(* CODESYS project twincat3_dioc_lib.library
   Author: AH
   Placeholder: Dioc
   Title: DiocLibrary
   Version: 3.25
   Company: Upzio

Project tree, tasks and I/O mapping:
  libraries: Tc2_Standard, * (Beckhoff Automation GmbH); Tc2_System, * (Beckhoff Automation GmbH); Tc2_Utilities, * (Beckhoff Automation GmbH); VisuDialogs, * (System)
  Data types/
    DIOC/
      Dioc/
        data type A_DIOC_DATA_TYPE
        data type A_DIOC_DATA_TYPE_1
        data type A_DIOC_MESSAGE
        data type A_DIOC_REGISTER_TYPE
        data type E_DIOC_ERROR
        data type E_DIOC_GEN_ERROR
        data type E_DIOC_REGISTER
        data type E_SM_DIOC
        data type E_SM_DIOC_DEVICE
        data type E_SM_DIOC_RECEIVE
        data type E_SM_DIOC_SEND
        data type ST_DIOC
        data type ST_DIOC_GEN_IN
        data type ST_DIOC_GEN_OUT
        data type ST_DIOC_IN
        data type ST_DIOC_LOG
        data type ST_DIOC_MESSINFO
        data type ST_DIOC_OUT
        data type ST_DIOC_REGISTER
      RC/
        RC/
          data type E_DIOC_RC_ERROR
          data type E_DIOC_RC_REGISTER
          data type E_RC_ERROR
          data type ST_DIOC_RC_IN
          data type ST_DIOC_RC_OUT
          data type ST_RC_IN
          data type ST_RC_OUT
      TP/
        TP10/
          data type E_DIOC_TP10_ERROR
          data type E_DIOC_TP10_REGISTER
          data type E_TP10
          data type E_TP10_ERROR
          data type ST_DIOC_TP10_IN
          data type ST_DIOC_TP10_OUT
          data type ST_TP10_IN
          data type ST_TP10_OUT
  Global Variables/
    global variables Global_DIOC_Constants
    global variables Global_DIOC_Variables
    global variables Global_DIOC_Variables_Debug
  POUs/
    DIOC/
      _Internal/
        DIOC/
          Dioc20/
            function F_DIOC_20_MESSAGE_IN [ST]
            function F_DIOC_20_MESSAGE_OUT [ST]
          function block FB_DIOC [ST]: Receive, Send, Startup
          function block FB_DIOC_GEN [ST]: Receive, Reset, Restart, Send, Startup
        DIOC_HELPFUNCTIONS/
          function F_DIOC_INC2 [ST]
          function F_DIOC_TO_DATE [ST]
          function F_SCALE_FROM_DIOC [ST]
          function F_SCALE_FROM_DIOC_FO [ST]
          function F_SCALE_FROM_REAL [ST]
          function F_SCALE_TO_DIOC [ST]
          function block FB_DIOC_FIFO [ST]
          function block FB_DIOC_RING [ST]
          function block FB_DIOC_RING2 [ST]
      RC/
        _Internal/
          function block FB_DIOC_RC [ST]: Receive, Restart, Send, Startup
          function block FB_RC_COMM [ST]: Startup
        function block FB_RC [ST]: StartupList, Stateinit
      TP10/
        _Internal/
          function block FB_DIOC_TP10 [ST]: Receive, Restart, Send, Startup
          function block FB_TP10_COMM [ST]: Startup
        function block FB_TP10 [ST]: StartupList, Stateinit
      function F_GetVersion_FIXSUS_DIOC [ST]
  Visualizations/
    DIOC/
      RC/
        RC_PARTS/
          visualisation RC_FP
          visualisation RC_ROOM_ICON
          visualisation UDO_DIPSWITCH
        visualisation RC
        visualisation RC_MINI
      TP10/
        TP10_PARTS/
          visualisation TP10_FP
          visualisation TP10_ROOM_ICON
        visualisation TP10
        visualisation TP10_MINI
  GlobalImagePool
*)

// Data types/DIOC/Dioc/A_DIOC_DATA_TYPE
TYPE A_DIOC_DATA_TYPE : DWORD;
END_TYPE

// Data types/DIOC/Dioc/A_DIOC_DATA_TYPE_1
TYPE A_DIOC_DATA_TYPE_1 : DWORD;
END_TYPE

// Data types/DIOC/Dioc/A_DIOC_MESSAGE
TYPE A_DIOC_MESSAGE : DWORD;
END_TYPE

// Data types/DIOC/Dioc/A_DIOC_REGISTER_TYPE
TYPE A_DIOC_REGISTER_TYPE : INT;
END_TYPE

// Data types/DIOC/Dioc/E_DIOC_ERROR
TYPE E_DIOC_ERROR :
(
	DIOC_ERROR_NO_ERROR
);
END_TYPE

// Data types/DIOC/Dioc/E_DIOC_GEN_ERROR
TYPE E_DIOC_GEN_ERROR :
(
	DIOC_REG_ERROR_NO_ERROR,
	DIOC_REG_ERROR_WRONG_TYPEID
);
END_TYPE

// Data types/DIOC/Dioc/E_DIOC_REGISTER
TYPE E_DIOC_REGISTER :
(
	DIOC_R00_SYNC_MESSAGE				:= 0,
	DIOC_R01_REGISTER_REQUEST			:= 1,
	DIOC_R02_REGISTER_INTERVAL			:= 2,
	DIOC_R03_TYPE_ID					:= 3,
	DIOC_R04_VERSION_HW					:= 4,
	DIOC_R05_VERSION_SW					:= 5,
	DIOC_R06_VERSION_REGISTERS			:= 6,
	DIOC_R07_UNIQUE_ID					:= 7,
	DIOC_R08_MESSAGE_ERROR_COUNTER		:= 8,
	DIOC_R09_VOLTAGE_LEVEL_A			:= 9,
	DIOC_R10_VOLTAGE_LEVEL_B			:= 10,
	DIOC_R11_DEVICE_ENABLE				:= 11,
	DIOC_R12_CPU_TEMPERATURE			:= 12,
	DIOC_R13_ErrorRegisterAdress		:= 13,

	DIOC_R84_TRANSMIT_DELAY				:= 84,
	DIOC_R85_SYNC_MESSAGE_HIGH			:= 85
);
END_TYPE

// Data types/DIOC/Dioc/E_SM_DIOC
TYPE E_SM_DIOC :
(
	SM_DIOC_POWERUP_DEVICE,					(* Activate device *)
	SM_DIOC_WAIT_FOR_DEVICE_CHARGED,		(* Activation timer, can be deactivated *)
	SM_DIOC_SEND_SYNC_REQUEST,				(* sync request by master *)
	SM_DIOC_WAIT_FOR_SYNC_ACK,				(* sync acknowledge by device *)
	SM_DIOC_SEND_SYNC_ACK,					(* sync acknowledge by master *)
	SM_DIOC_SEND_STARTUP_VALUES,			(* OPTIONAL Send optional startup values *)
	SM_DIOC_SEND_NEXTSTARTUP_VALUES,		(* OPTIONAL Send optional startup values *)
	SM_DIOC_R11_DEVICE_ENABLE,				(* OPTIONAL Enable Device *)
	SM_DIOC_R11_DEVICE_ENABLED,				(* OPTIONAL Enable Device *)
	SM_DIOC_ACTIVE				:= 100,		(* device is active *)
	SM_DIOC_END,
	SM_DIOC_TEST,
	SM_DIOC_WAIT_FOR_RESTART,				(* Delay time to restart after device failure *)
	SM_DIOC_ERROR 				:=666
);
END_TYPE

// Data types/DIOC/Dioc/E_SM_DIOC_DEVICE
TYPE E_SM_DIOC_DEVICE :
(
	SM_DIOC_DEVICE_POWERUP_DEVICE,					(* Power up device *)
	SM_DIOC_DEVICE_SEND_SYNC_REQUEST,				(* sync message by master *)
	SM_DIOC_DEVICE_SEND_SECOND_SYNC_REQUEST,		(* sync request by master *)
	SM_DIOC_DEVICE_WAIT_FOR_TYPE_ID,				(* wait until the device sent it's type id *)
	SM_DIOC_DEVICE_SEND_SYNC_ACK,					(* sync acknowledge by master *)
	SM_DIOC_DEVICE_SEND_STARTUP_VALUES,				(* OPTIONAL Send optional startup values *)
	SM_DIOC_DEVICE_STARTUP_VALUES_SENT,				(* OPTIONAL startup values sent *)
	SM_DIOC_DEVICE_DEVICE_ENABLE,					(* OPTIONAL Enable Device *)
	SM_DIOC_DEVICE_DEVICE_ENABLED,					(* OPTIONAL Enable Device *)
	SM_DIOC_DEVICE_RESTART,							(* device was restarted, wait until alle settings are re-written *)
	SM_DIOC_DEVICE_ACTIVE					:= 100,	(* device is active *)
	SM_DIOC_DEVICE_END,
	SM_DIOC_DEVICE_TEST,
	SM_DIOC_DEVICE_ERROR 					:= 666
);
END_TYPE

// Data types/DIOC/Dioc/E_SM_DIOC_RECEIVE
TYPE E_SM_DIOC_RECEIVE :
(
	SM_DIOC_RECEIVE_WAIT_FOR_DEVICE,
	SM_DIOC_RECEIVE_WAIT_FOR_STARTBIT,
	SM_DIOC_RECEIVE_RECEIVE_BITS,
	SM_DIOC_RECEIVE_WAIT_FOR_BUFFER,
	SM_DIOC_RECEIVE_END,
	SM_DIOC_RECEIVE_TEST,
	SM_DIOC_RECEIVE_ERROR	:= 666
);
END_TYPE

// Data types/DIOC/Dioc/E_SM_DIOC_SEND
TYPE E_SM_DIOC_SEND :
(
	SM_DIOC_SEND_WAIT_FOR_DEVICE,
	SM_DIOC_SEND_START,
	SM_DIOC_SEND_BITS,
	SM_DIOC_SEND_END,
	SM_DIOC_SEND_TEST,
	SM_DIOC_SEND_ERROR 			:=666
);
END_TYPE

// Data types/DIOC/Dioc/ST_DIOC
TYPE ST_DIOC :
STRUCT
	in						: ST_DIOC_IN;
	out						: ST_DIOC_OUT;
END_STRUCT
END_TYPE

// Data types/DIOC/Dioc/ST_DIOC_GEN_IN
TYPE ST_DIOC_GEN_IN :
STRUCT
	(* COMMANDS to device, bit reset by device block as an acknowledge *)
	(*Send start parameter*)

	bRxx_StartPar						: BOOL;

	(* Send test message *)
	bRxx_SendMessage					: BOOL;
	(* Send sync message *)
	bR00_SyncMessage					: BOOL;
	(* Register 1 / 2: register request *)
	bR01_RegisterRequest				: BOOL;
	bR01_RegisterRequestAutoSend		: BOOL;
	(* Sync delay *)
	bR84_TransmitDelay_READ				: BOOL;
	bR84_TransmitDelay_WRITE			: BOOL;

	(* COMMANDS to device, device uses the bit but does not alter it, eg output is switched when bit high, switched off when bit low *)
	bR03_Request_Type_ID				: BOOL;						(* R03: Type ID of the device *)
	bR04_Request_HW_Version				: BOOL;						(* R04: Hardware version of the device *)
	bR05_Request_SW_Version				: BOOL;						(* R05: Software version of the device *)
	bR06_Request_Register_Version		: BOOL;						(* R06: Register version of the device *)
	bR07_Request_Unique_ID				: BOOL;						(* R07: Unique ID of the device *)
	bR08_Message_Error_Counter_READ		: BOOL;						(* R08: message error counter *)
	bR08_Message_Error_Counter_WRITE	: BOOL;						(* R08: message error counter reset *)
	bR09_Read_DiocA_Voltage_Level		: BOOL;						(* R09: Read DIOCA voltage level (x10) *)
	bR10_Read_DiocB_Voltage_Level		: BOOL;						(* R10: Read DIOCB voltage level (x10) *)
	bR11_Enable_Device_READ				: BOOL;						(* R11: Device Enable *)
	bR11_Enable_Device					: BOOL;						(* R11: Device Enable *)
	bR11_Disable_Device					: BOOL;						(* R11: Device Disable *)
	bR12_CPU_Temperature				: BOOL;						(* R12: CPU Temperature *)

	(* DIOC OUTPUT PARAMETERS, parameters necessary for the above commands *)
	(* Send test message *)
	byRxx_SendMessageRegister 			: A_DIOC_REGISTER_TYPE	;	(* register address not inverted *)
	dwRxx_SendMessageData 				: A_DIOC_DATA_TYPE	:= 2#10;		(* data not inverted *)
	(* Register 1 / 2: register request *)
	dwR01_MessageRegister 				: A_DIOC_DATA_TYPE	;	(* register address not inverted *)
	dwR02_MessageAutoSendInterval		: A_DIOC_DATA_TYPE	:= 0;	(* 10 bit in seconds *)
	nR08_MessageErrorCounter			: UINT := 0;				(* R8: Message Err. Counter, onnly to be set <> 0 for unittest *)
	(* Sync delay *)
	dwR84_TransmitDelay					: A_DIOC_DATA_TYPE;
END_STRUCT
END_TYPE

// Data types/DIOC/Dioc/ST_DIOC_GEN_OUT
TYPE ST_DIOC_GEN_OUT :
STRUCT
	bDeviceActive					: BOOL;						(* Device is active *)
	(* Buffer statusses
	bRxBufferEmpty					: BOOL;						(* RX Buffer empty *)
	bRxBufferFull					: BOOL;						(* RX Buffer full *)
	bTxBufferEmpty					: BOOL;						(* All TX Buffer empty *)
	bTxBufferFull					: BOOL;						(* At least 1 TX Buffer full *)*)

	(* Internal feedback *)
	bTEST_LastMessageOK_Test		: BOOL;
	bRxx_Received					: BOOL;						(* There was a new message from the device *)

	(* RC register feedback bits *)
	bR11_DeviceEnabled				: BOOL;						(* R11: Device Enable *)

	(* RC register feedback values *)
	nRxx_Received					: INT;						(* There was a new message from the device from this register *)
	nR03_TypeID						: INT;						(* R3: Type ID *)
	nR08_MessageErrorCounter		: UINT;						(* R8: Message Err. Counter *)
	nR09_DiocVoltageA				: REAL := -3.402823E38; 	(* R9: Read DIOCA voltage level (x10) *)
	nR10_DiocVoltageB				: REAL := -3.402823E38; 	(* R10: Read DIOCA voltage level (x10) *)
	nR12_CpuTemperature				: REAL := -3.402823E38; 	(* R12: CPU Temperature *)
	nR13_ErrorRegisterAdress		: UINT;
	sR13_DtLastError				: STRING;
	nR84_TransmitDelay				: REAL := -3.402823E38;		(* R84: 'transmit delay (timeshift PLC<-> device) *)
	dtR04_VersionHW					: DATE;						(* R4: Version HW, 7 scrolls *)
	dtR05_VersionSW					: DATE;						(* R5: Version SW, 7 scrolls *)
	dtR06_VersionREG				: DATE;						(* R6: Version Registers, 7 scrolls *)
	sR07_UniqueID					: STRING[24];				(* R7: Unique ID *)
END_STRUCT
END_TYPE

// Data types/DIOC/Dioc/ST_DIOC_IN
TYPE ST_DIOC_IN :
STRUCT
	bEnable					: BOOL := TRUE;			(* TRUE powers the device *)
END_STRUCT
END_TYPE

// Data types/DIOC/Dioc/ST_DIOC_LOG
TYPE ST_DIOC_LOG :
STRUCT
	Message:ST_DIOC_REGISTER;
	Timestamp:DT;
	iArrId:INT;
END_STRUCT
END_TYPE

// Data types/DIOC/Dioc/ST_DIOC_MESSINFO
TYPE ST_DIOC_MESSINFO :
STRUCT
	nRegister							: A_DIOC_REGISTER_TYPE;
	nValue								: A_DIOC_DATA_TYPE;
	dt_Time								: DATE_AND_TIME;
	ArrnumberDIOC						: INT;
	iErrCode							: INT;
	iDeviceType							: INT;
END_STRUCT
END_TYPE

// Data types/DIOC/Dioc/ST_DIOC_OUT
TYPE ST_DIOC_OUT :
STRUCT
	bDeviceReady					: BOOL;				(* Device charged and ready *)
	(* DIOC Buffer statusses *)
	bRxBufferEmpty					: BOOL;				(* RX Buffer empty *)
	bRxBufferFull					: BOOL;				(* RX Buffer full *)
	bTxBufferEmpty					: BOOL;				(* All TX Buffer empty *)
	bTxBufferFull					: BOOL;				(* At least 1 TX Buffer full *)
	bBusyReceiving					: BOOL;			(* Receiving new data  *)
	bBusySending					: BOOL;				(* Sending data *)
	bError							: BOOL;				(* Dioc error state *)
	nErrorID						: E_DIOC_ERROR;		(* Dioc error code *)
	dwDataReceived					: DWORD;			(* Data received *)
END_STRUCT
END_TYPE

// Data types/DIOC/Dioc/ST_DIOC_REGISTER
TYPE ST_DIOC_REGISTER :
STRUCT
	nPLC_Cycle			: WORD;		(* Only for debugging *)
	nRegister			: A_DIOC_REGISTER_TYPE;
	nValue				: A_DIOC_DATA_TYPE;
END_STRUCT
END_TYPE

// Data types/DIOC/RC/RC/E_DIOC_RC_ERROR
TYPE E_DIOC_RC_ERROR :
(
	DIOC_RC_ERROR_NO_ERROR
);
END_TYPE

// Data types/DIOC/RC/RC/E_DIOC_RC_REGISTER
TYPE E_DIOC_RC_REGISTER :
(
	RC_R20_RC_TEMPERATURE			:= 20,
	RC_R21_PS_AC_VOLTAGE_LEVEL,
	RC_R22_STATUS_BITS_DIPSWITCHES,
	RC_R25_HEATING_7_8_3P			:= 25,
	RC_R26_HEATING_9_SP,
	RC_R27_HEATING_12_13_TEMP_HVAC_WATER,
	RC_R32_COOLING_20_21_3P		:= 32,
	RC_R33_COOLING_22_SP,
	RC_R34_COOLING_25_26_TEMP_ICE_WATER,
	RC_R39_PULSION_16_POSITION_COMMAND := 39,
	RC_R40_PULSION_17_POSITION_FEEDBACK,
	RC_R42_PULSION_18_AIR_TEMPERATURE := 42,
	RC_R45_EXTRACTION_29_POSITION_COMMAND := 45,
	RC_R46_EXTRACTION_30_POSITION_FEEDBACK,
	RC_R49_EXTRACTION_31_AIR_TEMPERATURE := 49,
	RC_R52_FIREDAMPER_33_34_COMMAND := 52,
	RC_R53_FIREDAMPER_36_37_FEEDBACK,
	RC_R56_FAN_39_40_SPEED_COMMAND 	:= 56,
	RC_R57_FAN_ENABLE,
	RC_R58_FAN_FAULT_STATUS,
	RC_R61_DO_45_46_47				:= 61,

	RC_R82_temperature_readout_adjust	:= 82,
	RC_R84_TRANSMIT_DELAY				:= 84,
	RC_R85_SYNC_MESSAGE_HIGH			:= 85
);
END_TYPE

// Data types/DIOC/RC/RC/E_RC_ERROR
TYPE E_RC_ERROR :
(
	RC_ERROR_NO_ERROR
);
END_TYPE

// Data types/DIOC/RC/RC/ST_DIOC_RC_IN
TYPE ST_DIOC_RC_IN :
STRUCT
	(* Startup list *)
	arrstStartupParameter				: ARRAY[1..DIOC_NOOFSTARTUPPARAMETERS] OF ST_DIOC_REGISTER;

	bR20_RC_Temperature				: BOOL;						(* R20: RC Temperature *)
	bR21_Read_PS_AC_Voltage				: BOOL;						(* R21: Read PS AC voltage level (x10) *)
	bR22_Status_Dip_Switches			: BOOL;						(* R22: Status bits DIP switches *)
	bR23_reserve						: BOOL;
	bR24_reserve						: BOOL;
	bR25_Heating_7_8_3p_plus_pwm		: BOOL;						(* R25: Heating 7-8 bit 0: 3p+/pwm, bit 1: 3p- *)
	bR25_Heating_7_8_3p_min				: BOOL;						(* R25: Heating 7-8 bit 0: 3p+/pwm, bit 1: 3p- *)
	bR25_Heating_7_8_3p_status			: BOOL;						(* R25: Heating 7-8 bit 0: 3p+/pwm, bit 1: 3p- *)
	bR26_Heating_SP						: BOOL;						(* R26: Heating 9  SP 0..10V *)
	bR26_Heating_SP_status				: BOOL;						(* R26: Heating 9  SP 0..10V *)
	bR27_Heating_T						: BOOL;						(* R27: Heating 12-13 temperature HVAC water *)
	bR28_reserve						: BOOL;
	bR29_reserve						: BOOL;
	bR30_reserve						: BOOL;
	bR31_reserve						: BOOL;
	bR32_Cooling_20_21_3p_plus_pwm		: BOOL;						(* R32: Cooling 20-21 bit 0: 3p+/pwm   1: 3p- *)
	bR32_Cooling_20_21_3p_min			: BOOL;						(* R32: Cooling 20-21 bit 0: 3p+/pwm   1: 3p- *)
	bR32_Cooling_20_21_3p_status		: BOOL;						(* R32: Cooling 20-21 bit 0: 3p+/pwm   1: 3p- *)
	bR33_Cooling_SP						: BOOL;						(* R33: Cooling 22  SP 0..10V *)
	bR33_Cooling_SP_status				: BOOL;						(* R33: Cooling 22  SP 0..10V *)
	bR34_Cooling_T						: BOOL;						(* R34: Cooling 25-26 temperature ICE water *)
	bR35_reserve						: BOOL;
	bR36_reserve						: BOOL;
	bR37_reserve						: BOOL;
	bR38_reserve						: BOOL;
	bR39_Pulsion_SP						: BOOL;						(* RC pulsion 16: 0..10V position command *)
	bR40_Pulsion_FB						: BOOL;						(* RC pulsion 17: 0..10V position feedback *)
	bR41_reserve						: BOOL;
	bR42_Pulsion_T						: BOOL;						(* RC pulsion 18-19 pulsion air temperature *)
	bR43_reserve						: BOOL;
	bR44_reserve						: BOOL;
	bR45_Extraction_SP					: BOOL;						(* RC extraction 29: 0..10V position command *)
	bR46_Extraction_FB					: BOOL;						(* RC extraction 30: 0..10V position feedback *)
	bR47_reserve						: BOOL;
	bR48_reserve						: BOOL;
	bR49_Extraction_T					: BOOL;						(* RC extraction 31-32 extraction air temperature *)
	bR50_reserve						: BOOL;
	bR51_reserve						: BOOL;
	bR52_FireDamperCOM_NO				: BOOL;						(* R52: FireDamper 33-34 bit 0: 2p NO   1: 2p NC  command *)
	bR52_FireDamperCOM_NC				: BOOL;						(* R52: FireDamper 33-34 bit 0: 2p NO   1: 2p NC  command *)
	bR52_FireDamperCOM_status			: BOOL;						(* R52: FireDamper 33-34 bit 0: 2p NO   1: 2p NC  command *)
	bR53_FireDamperCOM_FB				: BOOL;						(* R53: FireDamper 36-37 bit 0: FB_CLS  1: FB_OPN feedback *)
	bR54_reserve						: BOOL;
	bR55_reserve						: BOOL;
	bR56_Fan_SP							: BOOL;						(* R56: FAN 39-40: 0..10V fanspeed command *)
	bR57_Fan_Enable						: BOOL;						(* R57: FAN Enable command *)
	bR58_Fan_Fault_Status				: BOOL;						(* R58: FAN Fault status *)
	bR61_do_45							: BOOL;
	bR61_do_46							: BOOL;
	bR61_do_47							: BOOL;

	(* DIOC OUTPUT PARAMETERS, parameters necessary for the above commands *)
	(* Send test message *)
	nR26_Heating_SP						: UINT := 0;				(* R26: Heating 9  SP 0..4095 = 0..10V *)
	nR33_Cooling_SP						: UINT := 0;				(* R33: Cooling 22 SP 0..4095 = 0..10V *)
	nR39_Pulsion_SP						: UINT := 0;				(* R39: RC pulsion 16: 0..10V position command SP 0..4095 = 0..10V *)
	nR45_Extraction_SP					: UINT := 0;				(* R45: RC extraction 29: 0..10V position command SP 0..4095 = 0..10V *)
	nR56_Fan_SP							: UINT := 0;				(* R56: FAN 39-40: 0..10V fanspeed command SP 0..4095 = 0..10V *)
END_STRUCT
END_TYPE

// Data types/DIOC/RC/RC/ST_DIOC_RC_OUT
TYPE ST_DIOC_RC_OUT :
STRUCT
	(* RC register feedback bits *)
	(* bR11_DeviceEnabled				: BOOL;						R11: Device Enable *)
	bR22_Dipswitch_S01				: BOOL;						(* R22: 9_100%, 7_open *)
	bR22_Dipswitch_S02				: BOOL;						(* R22: 8_close *)
	bR22_Dipswitch_S03				: BOOL;						(* R22: 22_100%, 20_open *)
	bR22_Dipswitch_S04				: BOOL;						(* R22: 21_close *)
	bR22_Dipswitch_S05				: BOOL;						(* R22: 16_100% *)
	bR22_Dipswitch_S06				: BOOL;						(* R22: 29_100% *)
	bR22_Dipswitch_S07				: BOOL;						(* R22: 33 *)
	bR22_Dipswitch_S08				: BOOL;						(* R22: 34 *)
	bR22_Dipswitch_S09				: BOOL;						(* R22: 39_100% *)
	bR22_Dipswitch_S10				: BOOL;						(* R22: free soft 1 *)
	bR22_Dipswitch_S11				: BOOL;						(* R22: free soft 2 *)
	bR22_Dipswitch_S12				: BOOL;						(* R22: free soft 3 *)
	bR25_Heating_7_8_3p_plus_pwm	: BOOL;						(* R25: Heating 7-8 bit 0: 3p+/pwm, bit 1: 3p- *)
	bR25_Heating_7_8_3p_min			: BOOL;						(* R25: Heating 7-8 bit 0: 3p+/pwm, bit 1: 3p- *)
	bR32_Cooling_20_21_3p_plus_pwm	: BOOL;						(* R32: Cooling 20-21 bit 0: 3p+/pwm   1: 3p- *)
	bR32_Cooling_20_21_3p_min		: BOOL;						(* R32: Cooling 20-21 bit 0: 3p+/pwm   1: 3p- *)
	bR52_FireDamperCOM_NO			: BOOL;						(* R52: FireDamper 33-34 bit 0: 2p NO   1: 2p NC  command *)
	bR52_FireDamperCOM_NC			: BOOL;						(* R52: FireDamper 33-34 bit 0: 2p NO   1: 2p NC  command *)
	bR53_FireDamperFB_CLS			: BOOL;						(* R53: FireDamper 36-37 bit 0: FB_CLS  1: FB_OPN feedback *)
	bR53_FireDamperFB_OPN			: BOOL;						(* R53: FireDamper 36-37 bit 0: FB_CLS  1: FB_OPN feedback *)
	bR57_Fan_Enable					: BOOL;						(* R57: FAN Enable command *)
	bR58_FanFaultStatus				: BOOL;
	bR61_do_45						: BOOL;
	bR61_do_46						: BOOL;
	bR61_do_47						: BOOL;



	(* RC register feedback values *)
	nR20_RCTemperature				: REAL := -3.402823E38;		(* R20: RC Temperature *)
	nR21_PsAcVoltageLevel			: REAL := -3.402823E38;		(* R21: Read PS AC voltage level (x10) *)
	nR26_Heating_SP					: REAL := -3.402823E38;		(* R26: Heating 9 SP 0..10V *)
	nR27_HeatingTempHvacWater		: REAL := -3.402823E38;		(* R27: Heating 12-13 temperature HVAC water *)
	nR33_Cooling_SP					: REAL := -3.402823E38;		(* R33: Cooling 22 SP 0..10V *)
	nR34_CoolingTempIceWater		: REAL := -3.402823E38;		(* R34: Cooling 25-26 temperature ICE water *)
	nR39_Pulsion_SP					: REAL := -3.402823E38;		(* R39: RC pulsion 16: 0..10V position command *)
	nR40_Pulsion_FB					: REAL := -3.402823E38;		(* R40: RC pulsion 17: 0..10V position feedback *)
	nR42_PulsionAirTemperature		: REAL := -3.402823E38;		(* R42: RC pulsion 18-19 pulsion air temperature *)
	nR45_Extraction_SP				: REAL := -3.402823E38;		(* R45: RC extraction 29: 0..10V position command *)
	nR46_Extraction_FB				: REAL := -3.402823E38;		(* R46: RC extraction 30: 0..10V position feedback *)
	nR49_ExtractionAirTemperature	: REAL := -3.402823E38;		(* R49: RC extraction 31-32 pulsion air temperature *)
	nR56_Fan_SP						: REAL := -3.402823E38;		(* R56: FAN 39-40: 0..10V fanspeed command *)
	sR22_Dipswitch					: STRING[12];				(* R22: dipswitches overview *)
END_STRUCT
END_TYPE

// Data types/DIOC/RC/RC/ST_RC_IN
TYPE ST_RC_IN :
STRUCT
	bEnable						: BOOL := TRUE;	(* TRUE powers the device *)
	DIOC_Gen					: ST_DIOC_GEN_IN;
	DIOC_RC						: ST_DIOC_RC_IN;
END_STRUCT
END_TYPE

// Data types/DIOC/RC/RC/ST_RC_OUT
TYPE ST_RC_OUT :
STRUCT
	DIOC_Gen					: ST_DIOC_GEN_OUT;
	DIOC_RC					: ST_DIOC_RC_OUT;
END_STRUCT
END_TYPE

// Data types/DIOC/TP/TP10/E_DIOC_TP10_ERROR
TYPE E_DIOC_TP10_ERROR :
(
	DIOC_TP10_ERROR_NO_ERROR
);
END_TYPE

// Data types/DIOC/TP/TP10/E_DIOC_TP10_REGISTER
TYPE E_DIOC_TP10_REGISTER :
(
	TP10_R19_CONFIGURATION_SETUP				:= 19,
	TP10_R20_ROOMTEMPERATURE_SETUP,
	TP10_R21_ROOMTEMPERATURE,
	TP10_R22_ROOM_HUMIDITY_SETUP,
	TP10_R23_ROOM_HUMIDITY,
	TP10_R24_CO2_SETUP,
	TP10_R25_CO2,
	TP10_R26_VOC_SETUP,
	TP10_R27_VOC,
	TP10_R28_VOC_BASELINE_L_SETUP,
	TP10_R29_VOC_BASELINE_H_SETUP,


	TP10_R34_ROOM_ILLUMINATION_SETUP			:= 34,
	TP10_R35_ROOM_ILLUMINATION_LUXL_VALUE,
	TP10_R36_ROOM_ILLUMINATION_LUXH_VALUE,
	TP10_R37_ROOM_ILLUMINATION_IRL_VALUE,
	TP10_R38_ROOM_ILLUMINATION_IRH_VALUE,


	TP10_R50_TOUCH_BUTTON_STATUS				:=50,
	TP10_R51_TOUCH_LED_STATUS,
	TP10_R52_TOUCH_LED_MASK,
	TP10_R53_LED_INTENSITY_MAX,
	TP10_R54_LED_INTENSITY_MIN,
	TP10_R55_LED_APPROACH_INTENSITY,
	TP10_R56_LED_OFF_DELAY,
	TP10_R57_HAPTIC_INTENSITY,
	TP10_R58_TICK_BUTTON_SETUP,
	TP10_R59_TICK_BUTTON_VALUE,
	TP10_R60_RGB_LED_SETUP,
	TP10_R61_RGB_MSB,
	TP10_R62_RGB_LSB,

	TP10_R82_TEMP_OFFSET						:= 82, (*old temperature offset register*)
	TP10_R83_BUTTON_SENSITIVITY					:= 83, (*button sensitivity register*)
	TP10_TRANSMIT_DELAY							:= 84,
	TP10_SYNC_MESSAGE_HIGH						:= 85,
	TP10_R86_TEMP_OFFSET						:= 86 (*new temperature offset register*)


);
END_TYPE

// Data types/DIOC/TP/TP10/E_TP10
TYPE E_TP10 :
(
	TP10_INIT,
	TP10_START_CALIBRATION,
	TP10_SET_LED,
	TP10_WAIT_STARTUP,
	TP10_RESET_LED,
	TP10_CALIBRATED
);
END_TYPE

// Data types/DIOC/TP/TP10/E_TP10_ERROR
TYPE E_TP10_ERROR :
(
	TP10_ERROR_NO_ERROR
);
END_TYPE

// Data types/DIOC/TP/TP10/ST_DIOC_TP10_IN
TYPE ST_DIOC_TP10_IN :
STRUCT
	(* Startup list *)
	arrstStartupParameter				: ARRAY[1..DIOC_NOOFSTARTUPPARAMETERS] OF ST_DIOC_REGISTER;

	(* TP10 requests *)
	bR19_Configuration_Setup			: BOOL;						(*contains all info about sensor availability*)
	bR20_Room_Temperature_Setup			: BOOL;
	bR21_Room_Temperature				: BOOL;						(* R21: Room Temperature *)
	bR22_Room_Humidity_Setup			: BOOL;
	bR23_Room_Humidity					: BOOL;						(* R23: Room Humidity *)
	bR24_CO2_Setup						: BOOL;						(* R24: CO2 setup *)
	bR25_CO2_Values						: BOOL;						(* R24: CO2 values *)
	bR26_VOC_Setup						: BOOL;						(* R25: VOC Setup *)
	bR27_VOC_Values						: BOOL;						(* R26: VOC Values *)
	bR28_VOC_Baseline_L_SEND			: BOOL;
	bR29_VOC_Baseline_H_SEND			: BOOL;
	bR28_VOC_Baseline_L_REQ				: BOOL;
	bR29_VOC_Baseline_H_REQ				: BOOL;
	bR34_LUX_Setup						: BOOL;
	bR35_LUX_L							: BOOL;
	bR36_LUX_H							: BOOL;
	bR37_IR_L							: BOOL;
	bR38_IR_H							: BOOL;



	bR51_TouchLedStatus					: BOOL;
	bR51_TouchLed01						: BOOL;						(* R51: switch touch LED *)
	bR51_TouchLed02						: BOOL;
	bR51_TouchLed03						: BOOL;
	bR51_TouchLed04						: BOOL;
	bR51_TouchLed05						: BOOL;
	bR51_TouchLed06						: BOOL;
	bR51_TouchLed07						: BOOL;
	bR51_TouchLed08						: BOOL;
	bR51_TouchLed09						: BOOL;
	bR51_TouchLed10						: BOOL;
	bR52_TouchLedMaskStatus				: BOOL;						(* R52: Retrieve touch LED mask status *)
	bR52_TouchLedMask01					: BOOL;						(* R52: Set individual touch LED mask touch xx *)
	bR52_TouchLedMask02					: BOOL;
	bR52_TouchLedMask03					: BOOL;
	bR52_TouchLedMask04					: BOOL;
	bR52_TouchLedMask05					: BOOL;
	bR52_TouchLedMask06					: BOOL;
	bR52_TouchLedMask07					: BOOL;
	bR52_TouchLedMask08					: BOOL;
	bR52_TouchLedMask09					: BOOL;
	bR52_TouchLedMask10					: BOOL;
	bR50_TouchButtonStatus				: BOOL;						(* R50: Retrieve touch button status *)
	bR57_HapticIntensity				: BOOL;						(* R57: Haptic Intensity write *)
	bR57_HapticIntensityStatus			: BOOL;						(* R57: Haptic Intensity read *)
	bR53_LED_Intensity_Max				: BOOL;
	bR54_LED_Intensity_Min				: BOOL;
	bR56_LED_Led_off_delay				: BOOL;



	nR60_RGB_LED_SETUP					: A_DIOC_DATA_TYPE := 0;
	nR61_RGB_MSB						: A_DIOC_DATA_TYPE := 0;
	nR62_RGB_LSB						: A_DIOC_DATA_TYPE := 0;

	nR61_RGB_RED						: BYTE;
	nR61_RGB_GREEN						: BYTE;
	nR61_RGB_BlUE						: BYTE;

	(* DIOC OUTPUT PARAMETERS, parameters necessary for the above commands *)


	nR20_ROOMTEMPERATURE_SETUP			: A_DIOC_DATA_TYPE:=1; (*LSB = 1 = sensor activated, 0 = no read, disabled*)
	nR21_ROOMTEMPERATURE				: REAL:=0; (* 0..2048 = -20°C..120°C *)
	nR22_ROOM_HUMIDITY_SETUP			: A_DIOC_DATA_TYPE:=1; (*LSB = 1 = sensor activated, 0 = no read, disabled*)
	nR23_ROOM_HUMIDITY					: REAL:=0; (* 0..2048 = 0..2048 ppm *)
	nR24_CO2_SETUP						: A_DIOC_DATA_TYPE:=1; (*LSB = 1 = sensor activated, 0 = no read, disabled*)
	nR25_CO2							: REAL:=0; (* 0..2048 = 0..2048 ppm *)
	nR26_VOC_SETUP						: A_DIOC_DATA_TYPE:=1; (*LSB = 1 = sensor activated, 0 = no read, disabled*)
	nR27_VOC							: REAL:=0; (* 0..2048 = 0..2048 ppm *)

	nR34_ROOM_ILLUMINATION_SETUP		: A_DIOC_DATA_TYPE:=1;
	nR35_ROOM_ILLUMINATION_LUXL_VALUE	: REAL:=0;
	nR36_ROOM_ILLUMINATION_LUXH_VALUE	: REAL:=0;
	nR37_ROOM_ILLUMINATION_IRL_VALUE	: REAL:=0;
	nR38_ROOM_ILLUMINATION_IRH_VALUE	: REAL:=0;

	nR50_TOUCH_BUTTON_STATUS			: A_DIOC_DATA_TYPE := 0;	(* R51: Touch LED status *)
	nR51_TouchLedStatus					: A_DIOC_DATA_TYPE := 0;	(* R51: Touch LED status *)
	nR52_TouchLedMask					: A_DIOC_DATA_TYPE := 1050;	(* R52: Touch LED mask, 1050 = all 10 leds active *)
	nR57_HapticIntensity				: A_DIOC_DATA_TYPE := 100;	(* R57: Haptic Intensity, in percentage *)
	nR53_LED_Intensity_Max				: A_DIOC_DATA_TYPE := 0;	(* R25: LED_L intensity, in percentage *)
	nR54_LED_Intensity_Min				: A_DIOC_DATA_TYPE := 0;	(* R26: LED_R intensity, in percentage *)

	NR82_Temp_offset					: A_DIOC_DATA_TYPE := 22;	(*  *)
	NR83_ButtonSensitivity				: A_DIOC_DATA_TYPE := 0;	(*button sensitivity*)
	NR86_Temp_offset					: A_DIOC_DATA_TYPE := 1484;	(**)
	bR82_Temp_offset					: BOOL; (*resend temperature offset if true*)
	bR86_Temp_offset					: BOOL; (*resend temperature offset if true*)
END_STRUCT
END_TYPE

// Data types/DIOC/TP/TP10/ST_DIOC_TP10_OUT
TYPE ST_DIOC_TP10_OUT :
STRUCT
	(* Calibration finished? *)
	bCalibrationFinished						: BOOL;
	(* TP10 register feedback bits *)
	(* Register 08 *)
	byR29_WaveDetected						: BYTE;						(* 0001 = minimum, 0010 = down, 0100 = up, 1000=maximum *)
	(* Register 03: Button status bits (bit 0-9) *)
	bR50_TouchButton01						: BOOL;
	bR50_TouchButton02						: BOOL;
	bR50_TouchButton03						: BOOL;
	bR50_TouchButton04						: BOOL;
	bR50_TouchButton05						: BOOL;
	bR50_TouchButton06						: BOOL;
	bR50_TouchButton07						: BOOL;
	bR50_TouchButton08						: BOOL;
	bR50_TouchButton09						: BOOL;
	bR50_TouchButton10						: BOOL;

	(* UNIT SENSORS *)
	(* Register 04: Room temperature *)

	nR51_TouchLedStatus						: A_DIOC_DATA_TYPE := 0;	(* R21: Touch LED status *)
	nR52_TouchLedMask						: A_DIOC_DATA_TYPE := 1023;	(* R22: Touch LED mask, 4095 = all active *)
	nR50_TouchButtonStatus					: A_DIOC_DATA_TYPE := 0;	(* R23: Touch BUTTON status *)

	nR19_CONFIGURATION_SETUP			: A_DIOC_DATA_TYPE := 0;

	nR19_ROOMTEMPERATURE_AVAILABLE 		: BOOL;
	nR19_HUMIDITY_AVAILABLE 			: BOOL;
	nR19_CO2_AVAILABLE 					: BOOL;
	nR19_VOC_AVAILABLE 					: BOOL;
	nR19_CO_AVAILABLE 					: BOOL;
	nR19_PRESSURE_AVAILABLE 			: BOOL;
	nR19_REFPRESSURE_AVAILABLE 			: BOOL;
	nR19_ILLUMINATION_AVAILABLE 		: BOOL;
	nR19_TOUCH_AVAILABLE 				: BOOL;
	nR19_PROXIMITY_AVAILABLE 			: BOOL;
	nR19_HAPTIC_AVAILABLE				: BOOL;
	nR19_RGB_AVAILABLE 					: BOOL;

	nR20_ROOMTEMPERATURE_SETUP			: REAL:=0; (*LSB = 1 = sensor activated, 0 = no read, disabled*)
	nR21_ROOMTEMPERATURE				: REAL:=0; (* 0..2048 = -20°C..120°C *)
	nR22_ROOM_HUMIDITY_SETUP			: REAL:=0; (*LSB = 1 = sensor activated, 0 = no read, disabled*)
	nR23_ROOM_HUMIDITY					: REAL:=0; (* 0..2048 = 0..100 % *)
	nR24_CO2_SETUP						: REAL:=0; (*LSB = 1 = sensor activated, 0 = no read, disabled*)
	nR25_CO2							: REAL:=0; (* 0..2048 = 0..2048 ppm *)
	nR26_VOC_SETUP						: REAL:=0; (*LSB = 1 = sensor activated, 0 = no read, disabled*)
	nR27_VOC							: REAL:=0; (* 0..2048 = 0..2048 ppm *)
	nR28_VOC_BASELINE_L_SETUP			: A_DIOC_DATA_TYPE:=0;
	nR29_VOC_BASELINE_H_SETUP			: A_DIOC_DATA_TYPE:=0;
	br29_VOC_BASELINE_VALID				: BOOL;

	nR34_ROOM_ILLUMINATION_SETUP		: REAL:=0;
	nR35_ROOM_ILLUMINATION_LUXL_VALUE	: REAL:=0;
	nR36_ROOM_ILLUMINATION_LUXH_VALUE	: REAL:=0;
	nR37_ROOM_ILLUMINATION_IRL_VALUE	: REAL:=0;
	nR38_ROOM_ILLUMINATION_IRH_VALUE	: REAL:=0;

END_STRUCT
END_TYPE

// Data types/DIOC/TP/TP10/ST_TP10_IN
TYPE ST_TP10_IN :
STRUCT
	bEnable						: BOOL := TRUE;	(* TRUE powers the device *)
	DIOC_Gen					: ST_DIOC_GEN_IN;
	DIOC_TP10					: ST_DIOC_TP10_IN;
END_STRUCT
END_TYPE

// Data types/DIOC/TP/TP10/ST_TP10_OUT
TYPE ST_TP10_OUT :
STRUCT
	DIOC_Gen					: ST_DIOC_GEN_OUT;
	DIOC_TP10					: ST_DIOC_TP10_OUT;
END_STRUCT
END_TYPE

// Global Variables/Global_DIOC_Constants
{attribute 'Tc2GvlVarNames'}
VAR_GLOBAL CONSTANT
(* contains all data that is constant for the DIOC system*)
	(* TP10 *)
	DIOC_NOOFSTARTUPPARAMETERS		: INT := 40;	(* No of startup parameters in dioc device *)
	DIOC_RXTX_BUFFERSIZE					: INT := 10;		(* Same size for RX and TX *)
	DIOC_MAXPRIORITY						: INT := 8;		(* Maximum priority level *)
	DIOC_INVALID_REGISTER					: INT := 255;	(* indicates an invalid register *)
	DIOC_MAXRINGBUFFERSIZE				: INT := 20;	(* Max size of the local dioc ringbuffers *)

	(* Default color definitions DIOC
		nFillColor := 16#1E8FE03F;
		?1E (30%): intensity in percentage (64h (100) = full on, 00 = off)
		?8F: red
		?E0: green
		?3F: blue*)
	RGB_BLACK 								: DWORD := 16#1E000000;
	RGB_NAVY 								: DWORD := 16#1E000080;
	RGB_BLUE 								: DWORD := 16#1E0000FF;
	RGB_GREEN 							: DWORD := 16#1E008000;
	RGB_TEAL 								: DWORD := 16#1E008080;
	RGB_LIME 								: DWORD := 16#1E00FF00;
	RGB_AQUA 								: DWORD := 16#1E00FFFF;
	RGB_MAROON 							: DWORD := 16#1E800000;
	RGB_PURPLE							: DWORD := 16#1E800080;
	RGB_OLIVE 								: DWORD := 16#1E808000;
	RGB_GREY  								: DWORD := 16#1E808080;
	RGB_SILVER 							: DWORD := 16#1EC0C0C0;
	RGB_RED 								: DWORD := 16#1EFF0000;
	RGB_ORANGE 							: DWORD := 16#1EFFA500;
	RGB_FUCHSIA							: DWORD := 16#1EFF00FF;
	RGB_YELLOW  							: DWORD := 16#1EFFFF00;
	RGB_WHITE 								: DWORD := 16#1EFFFFFF;

END_VAR

// Global Variables/Global_DIOC_Variables
{attribute 'Tc2GvlVarNames'}
VAR_GLOBAL
(* contains all general dioc information and arrays *)
	DIOC_bRestart 					: BOOL;

(* timer that prevents all DIOC devices to start at the same time *)
	DIOC_tonLastStart 					: TON ;

(* -------> ONLY NECESSARY FOR INTERNAL DEBUGGING *)
	(* Time string for DIOC error log
	OPTIONAL: The DIOC devices need the system time as a string to do internal timestamping,
	if for debugging reasons the exact time must be logged, it must be set in gv_dioc_sSystemTimeString
	Can be any content, but must be a string of MAX 23	*)
	gv_dioc_sSystemTimeString		: STRING(23) := '';	 (*e.g.  2011_11_23__15h23m22s  *)

(* buffer that keeps track of all incoming and outgoing data of the analysed device*)
	DIOC_RECEIVE_LOG				: ARRAY[0..DIOC_MAXRINGBUFFERSIZE] OF ST_DIOC_REGISTER;
	DIOC_SEND_LOG					: ARRAY[0..DIOC_MAXRINGBUFFERSIZE] OF ST_DIOC_REGISTER;
END_VAR

// Global Variables/Global_DIOC_Variables_Debug
{attribute 'Tc2GvlVarNames'}
VAR_GLOBAL
(* !!!! Do not remove from the library !!!! *)
(* Variables for the Debug screen *)
	DIOC_DEBUG_SCREEN_ACTIVE	: BOOL := FALSE; (* Enable the button analyze *)
	DIOC_DEBUGLINKPREVSCREEN	: STRING[40] 	:= 'TC_VISU';
	DIOC_DEBUGSCHERM			: STRING[40] 	:= 'DIOC_DEBUG'; (*name visualisation analyse screen*)
	DIOC_Debug 						: BOOL		:=	FALSE; (*Do not make this true if the analyse screen isn't being used*)
	DIOC_pDebugged_TP10			: POINTER TO FB_TP10; (*pointer to the analysed TP10 device*)
	DIOC_pDebugged_RC				: POINTER TO FB_RC; (*pointer to the analysed RC device*)
(* ONLY NECESSARY FOR INTERNAL DEBUGGING <------- *)
END_VAR

// POUs/DIOC/_Internal/DIOC/Dioc20/F_DIOC_20_MESSAGE_IN
(*
	Breaks down the dioc message in a register and a data part *)
FUNCTION F_DIOC_20_MESSAGE_IN : ST_DIOC_REGISTER
VAR_INPUT
	IN				: A_DIOC_MESSAGE;
END_VAR
VAR
END_VAR

(*
	Filter the register *)
F_DIOC_20_MESSAGE_IN.nRegister			:= 127 - DWORD_TO_BYTE(ROR(IN AND 2#1111111_0, 1));

(*
	Filter the data *)
F_DIOC_20_MESSAGE_IN.nValue			:= 4095 - ((IN / 256) AND 2#1111_1111_1111);

END_FUNCTION

// POUs/DIOC/_Internal/DIOC/Dioc20/F_DIOC_20_MESSAGE_OUT
(*Combines register and a data part to a dioc message *)
FUNCTION F_DIOC_20_MESSAGE_OUT : A_DIOC_MESSAGE
VAR_INPUT
	nRegister			: A_DIOC_REGISTER_TYPE;
	nValue				: A_DIOC_DATA_TYPE;
END_VAR
VAR
	bitRegister			: WORD;
	bitValue			: DWORD;
END_VAR

(*End, Bit 21 *)
bitValue 		:= (4095 - MIN(nValue,4095)) * 256;	(* Shift inverted data 8 bits *)
bitRegister		:= INT_TO_WORD((127 - nRegister) * 2);	(* Shift inverted data 1 bit, first bit is always 0 *)
F_DIOC_20_MESSAGE_OUT			:= 1048576;	(* first bit at position 21, last bit is always 1 *)
F_DIOC_20_MESSAGE_OUT			:= F_DIOC_20_MESSAGE_OUT + bitValue;
F_DIOC_20_MESSAGE_OUT			:= F_DIOC_20_MESSAGE_OUT + bitRegister;

END_FUNCTION

// POUs/DIOC/_Internal/DIOC/FB_DIOC
(*
	General dioc communication block *)
FUNCTION_BLOCK FB_DIOC
VAR_INPUT
	(* Data handshake interface *)
	in									: ST_DIOC_IN;
	(* Dioc device specific constants *)
	DEVICE_CHARGE_TIME					: TIME 		:= T#2s;			(* ICU: if extra time is needed *)
	DIOC_LENGTH							: INT 		:= 21;				(* DIOC protocol length *)

	iPowerCycleGroup					: INT;
END_VAR
VAR_OUTPUT
	(* Dioc feedback data *)
	Out									: ST_DIOC_OUT;
END_VAR
VAR_IN_OUT
	(* Message buffers *)
	RxBuffer							: ARRAY[0..DIOC_RXTX_BUFFERSIZE] OF A_DIOC_MESSAGE;	(* 1 message queue *)
	TxBuffer							: ARRAY[0..DIOC_MAXPRIORITY, 0..DIOC_RXTX_BUFFERSIZE] OF A_DIOC_MESSAGE;	(* 1 message queue / priority, HIGHEST: 0 = internal priority *)
	(* Fifo Buffer handlers *)
	fbRxBuffer							: FB_DIOC_FIFO;								(* 1 message queue *)
	fbTxBuffer							: ARRAY[0..DIOC_MAXPRIORITY] OF FB_DIOC_FIFO;	(* 1 message queue / priority *)
END_VAR
(*
	local dioc constants *)
VAR CONSTANT
	OUT_LEVEL_HIGH						: BOOL := FALSE;
	OUT_LEVEL_LOW						: BOOL := TRUE;
	IN_LEVEL_HIGH						: BOOL := FALSE;
	IN_LEVEL_LOW						: BOOL := TRUE;
	TIMEOUT_RECEIVE_OFF					: TIME := T#1s;
	TIMEOUT_RECEIVE_ON					: TIME := T#1m;
END_VAR
VAR
(* TC3 attribute, will be ignored by TC2 *)
{attribute 'hide_all_locals'}
(* TC2 attribute, will be ignored by TC3 *)
{library private}
	(* IO *)
	diIn						AT 	%I*	: BOOL;
	doOut						AT 	%Q*	: BOOL;

	(* State machines *)
	nSm									: E_SM_DIOC;
	nSmReceive							: E_SM_DIOC_RECEIVE;
	nSmSend								: E_SM_DIOC_SEND;

	(* Rx / Tx logging Ring buffers *)
	fbDioc_Ring_Rx						: FB_DIOC_RING;
	fbDioc_Ring_Tx						: FB_DIOC_RING;

{library private}
	(* Timers *)
	tTimerStartup						: TON;
	tReceiveTimeout						: TON;
	tDeviceFailureDiOff					: TON;
	tDeviceFailureDiOn					: TON;

	(* Messages *)
	nMessageSend						: DWORD;
	nMessageReceive						: DWORD;
	nMessageSendPointer					: INT;
	nMessageReceivePointer				: INT;

	(*
		Startup *)
	bStartup							: BOOL := TRUE;

	(*
		Which buffer (sorted highest priority) has data to be sent *)
	nTxBufferContainsItems				: INT;			(* next tx buffer to be treated *)
	i									: INT;

	(*
		Buffer read / write *)
	bRxBuffer_Read						: BOOL;
	bRxBuffer_Write						: BOOL;
	bTxBuffer_Read						: BOOL;
	bTxBuffer_Write						: BOOL;

	(*
		Ring buffer write *)
	Dioc_Register						: ST_DIOC_REGISTER;		(* Message for ring buffer *)
	bRxRingBuffer_Write					: BOOL;
	bTxRingBuffer_Write					: BOOL;

	(* Debugging pointer, increments every plc cycle, to see when the messages were sent *)
	nPLC_Cycle							: WORD;
END_VAR

(*
	startup *)
IF bStartup THEN Startup(); END_IF

(* Debugging pointer, increments every plc cycle, to see when the messages were sent *)
nPLC_Cycle := nPLC_Cycle + 1;

(*
	Startup timer, charging of the capacitors of the device *)
tTimerStartup(IN:= (nSm = SM_DIOC_WAIT_FOR_DEVICE_CHARGED), PT:= DEVICE_CHARGE_TIME, Q=> , ET=> );

(*
	timeout Receive, if nothing was received for a long time *)
tReceiveTimeout(IN := (nSmReceive = SM_DIOC_RECEIVE_WAIT_FOR_STARTBIT), PT:= TIMEOUT_RECEIVE_OFF, Q=> , ET=> );

(*
	The device dropped the input too long, something must be wrong, restart it *)
tDeviceFailureDiOff(IN := (nSm = SM_DIOC_ACTIVE AND NOT diIn) OR (nSm = SM_DIOC_WAIT_FOR_RESTART), PT:= TIMEOUT_RECEIVE_OFF, Q=> , ET=> );
tDeviceFailureDiOn(IN := (nSm = SM_DIOC_ACTIVE AND diIn) OR (nSm = SM_DIOC_WAIT_FOR_RESTART), PT:= TIMEOUT_RECEIVE_ON, Q=> , ET=> );

(*
	Receive *)
Receive();

(*
	General state machine *)
(* Device deactivated? => reset state machine *)
IF NOT in.bEnable 				THEN
	doOut 						:= in.bEnable;		(* If TRUE sets power to the device *)
	nSm 						:= SM_DIOC_POWERUP_DEVICE;
	nSmSend						:= SM_DIOC_SEND_WAIT_FOR_DEVICE;
	nSmReceive					:= SM_DIOC_RECEIVE_WAIT_FOR_DEVICE;
END_IF

CASE nSm	OF
	SM_DIOC_POWERUP_DEVICE:				(* Activate device *)
		(* 	ENABLE / DISABLE DEVICE *)
		(*	ONLY AT INITIAL STARTUP OR TIMEOUT
			as long as there is no connection made by the device remain in this step  
			connection is assumed when there is positive voltage detected since this is the only way to be sure the device is alive *)
		IF in.bEnable (*AND (gv_iPowerCycle = iPowerCycleGroup)*)  THEN
			doOut 			:= in.bEnable;		(* If TRUE sets power to the device *)
		ELSE
			doOut 			:= FALSE;		(* If TRUE sets power to the device *)
		END_IF

		out.bDeviceReady				:= FALSE;		(* Device is not ready *)
		IF diIn	 AND doOut 				THEN	(* Device signals enabled and is still enabled by upper level *)
			nSm 						:= SM_DIOC_WAIT_FOR_DEVICE_CHARGED;
		END_IF

	SM_DIOC_WAIT_FOR_DEVICE_CHARGED:	(* Activation timer, can be deactivated *)
		(* Give the device the opportunity to load the capacitors before sending the first message *)
		IF tTimerStartup.Q 				THEN
			fbDioc_Ring_Rx.RST 			:= TRUE;
			fbDioc_Ring_Tx.RST 			:= TRUE;
			nSm 						:= SM_DIOC_ACTIVE;
		END_IF

	SM_DIOC_ACTIVE:						(* device is active *)
		out.bDeviceReady				:= TRUE;		(* Device reaction, device is ready *)
		IF tDeviceFailureDiOff.Q OR tDeviceFailureDiOn.Q	THEN
			tDeviceFailureDiOff(IN := FALSE);	(* Reset timer *)
			tDeviceFailureDiOn(IN := FALSE);	(* Reset timer *)
			nSm 						:= SM_DIOC_WAIT_FOR_RESTART;
		END_IF

	SM_DIOC_END:
		;

	SM_DIOC_WAIT_FOR_RESTART:
		IF tDeviceFailureDiOff.Q OR tDeviceFailureDiOn.Q	THEN
			nSm							:= SM_DIOC_POWERUP_DEVICE;
		END_IF

	SM_DIOC_TEST:
		;

	SM_DIOC_ERROR:
		;

END_CASE

(*
	Send *)
Send();

(*
	Buffer status feedback, must be set BEFORE fb calls 
bRxBufferFull				:= out.bRxBufferFull;
bRxBufferEmpty				:= fbDioc.bRxBufferEmpty;
bTxBufferFull				:= fbDioc.bTxBufferFull;
bTxBufferEmpty				:= fbDioc.bTxBufferEmpty; *)

(*
	First loop finished *)
bStartup 					:= FALSE;

ACTION Receive:
(*
	Receive state machine *)
CASE nSmReceive 	OF

	SM_DIOC_RECEIVE_WAIT_FOR_DEVICE:;
		(* 	Wait until the device has powered up *)
		out.bBusyReceiving			:= FALSE;
		IF (nSm > SM_DIOC_WAIT_FOR_DEVICE_CHARGED) THEN
			nSmReceive := SM_DIOC_RECEIVE_WAIT_FOR_STARTBIT;
		END_IF

	SM_DIOC_RECEIVE_WAIT_FOR_STARTBIT:
		(* Wait for a new message *)
		out.bBusyReceiving			:= FALSE;
		IF (nSm <= SM_DIOC_WAIT_FOR_DEVICE_CHARGED) THEN
			nSmReceive 				:= SM_DIOC_RECEIVE_WAIT_FOR_DEVICE;
		ELSIF diIn	= IN_LEVEL_HIGH 	THEN
			out.bBusyReceiving		:= TRUE;
			nMessageReceive 		:= 0;		(* Reset received message *)
			nMessageReceive.0 		:= diIn;	(* Register first bit *)
			nMessageReceivePointer 	:= 1;
			nSmReceive				:= SM_DIOC_RECEIVE_RECEIVE_BITS;
		END_IF

	SM_DIOC_RECEIVE_RECEIVE_BITS:
		nMessageReceive.0 			:= diIn;
		nMessageReceivePointer 		:= nMessageReceivePointer + 1;
		(* Complete message received? *)
		IF nMessageReceivePointer < DIOC_LENGTH THEN
			nMessageReceive 		:= ROR(nMessageReceive,1);
		ELSE
			nMessageReceive 		:= ROR(nMessageReceive,33-DIOC_LENGTH);
			(* Shift the message to the receive buffer, goto wait step if the buffer is full *)
			IF fbRxBuffer.FULL		THEN
				nSmReceive			:= SM_DIOC_RECEIVE_WAIT_FOR_BUFFER;
			ELSE
				fbRxBuffer.IN		:= nMessageReceive;
				bRxBuffer_Write		:= TRUE;
				IF (nSm > SM_DIOC_WAIT_FOR_DEVICE_CHARGED) THEN
					nSmReceive := SM_DIOC_RECEIVE_WAIT_FOR_STARTBIT;
				ELSE
					nSmReceive 		:= SM_DIOC_RECEIVE_WAIT_FOR_DEVICE;
				END_IF
			END_IF
		END_IF

	SM_DIOC_RECEIVE_WAIT_FOR_BUFFER:
		(* Shift the message to the receive buffer, wait if the buffer is not full *)
		IF NOT fbRxBuffer.FULL		THEN
			fbRxBuffer.IN			:= nMessageReceive;
			bRxBuffer_Write			:= TRUE;
			IF (nSm > SM_DIOC_WAIT_FOR_DEVICE_CHARGED) THEN
				nSmReceive 			:= SM_DIOC_RECEIVE_WAIT_FOR_STARTBIT;
			ELSE
				nSmReceive 			:= SM_DIOC_RECEIVE_WAIT_FOR_DEVICE;
			END_IF
		END_IF

	SM_DIOC_RECEIVE_END:;

	SM_DIOC_RECEIVE_TEST:;

	SM_DIOC_RECEIVE_ERROR:;

	ELSE;

END_CASE

(* Log to ringbuffer? *)
bRxRingBuffer_Write := bRxBuffer_Write;

(*
	Message queue *)
fbRxBuffer(
	fifo		:= ADR(RxBuffer),
	RD			:= bRxBuffer_Read,
	WD			:= bRxBuffer_Write,
	EMPTY		=> out.bRxBufferEmpty,
	FULL		=> out.bRxBufferFull,
	);

(* Log to ringbuffer *)
bRxRingBuffer_Write := bRxRingBuffer_Write AND NOT bRxBuffer_Write; (* correctly written *)
Dioc_Register := F_DIOC_20_MESSAGE_IN(fbRxBuffer.IN);
fbDioc_Ring_Rx(
	nPLC_Cycle 	:= nPLC_Cycle,
	IN			:= Dioc_Register,
	WD			:= bRxRingBuffer_Write
	);
END_ACTION

ACTION Send:
(*
	Evaluate Message queue *)
nTxBufferContainsItems 				:= -1;
out.bTxBufferEmpty					:= TRUE;
out.bTxBufferFull					:= FALSE;
FOR i := DIOC_MAXPRIORITY TO 0 BY -1 DO
	(*	Is there a value in queue, highest priority buffer no is returned *)
	IF NOT fbTxBuffer[i].EMPTY 		THEN
		out.bTxBufferEmpty			:= FALSE;
		nTxBufferContainsItems 		:= i;
		(* Is it full ? *)
		IF fbTxBuffer[i].FULL		THEN
			out.bTxBufferFull		:= TRUE;
		END_IF
	END_IF
END_FOR

(*
	Send state machine *)
CASE nSmSend 	OF

	SM_DIOC_SEND_WAIT_FOR_DEVICE:
		(* 	Wait until the device has powered up *)
		out.bBusySending			:= FALSE;
		IF (nSm > SM_DIOC_WAIT_FOR_DEVICE_CHARGED) THEN
			nSmSend := SM_DIOC_SEND_START;
		END_IF

	SM_DIOC_SEND_START:
		(*	Give possibility to disable the device
			Check if too many messages have been sent in a row, generate delay before sending new commands 
			Wait for command to start the device 
			Wait for timeout if long time nothing has been sent *)
		out.bBusySending			:= FALSE;
		IF (nSm <= SM_DIOC_WAIT_FOR_DEVICE_CHARGED) THEN
			nSmSend 				:= SM_DIOC_SEND_WAIT_FOR_DEVICE;
		ELSIF nTxBufferContainsItems > -1	THEN
			out.bBusySending		:= TRUE;
			(* Fetch the next value from the fifo buffer *)
			bTxBuffer_Read			:= TRUE;
			fbTxBuffer[nTxBufferContainsItems](
				RD		:= bTxBuffer_Read,
				WD		:= bTxBuffer_Write,
				fifo	:= ADR(TxBuffer[nTxBufferContainsItems, 0])
				);
			bTxRingBuffer_Write 	:= TRUE; (* Log to ringbuffer *)
			(*	Combine register + data TO message *)
			nMessageSend      		:= fbTxBuffer[nTxBufferContainsItems].OUT;		(* message from the fifo register *)
			(* Start sending messsage *)
			doOut					:= nMessageSend.0;
			nMessageSend 			:= ROR(nMessageSend,1);
			nMessageSendPointer 	:= 1;	(* Reset pointer *)
			nSmSend					:= SM_DIOC_SEND_BITS;
		END_IF

	SM_DIOC_SEND_BITS:
		(* Send all bits of the message *)
		doOut						:= nMessageSend.0;
		nMessageSend 				:= ROR(nMessageSend,1);
		nMessageSendPointer 		:= nMessageSendPointer + 1;
		IF nMessageSendPointer		 >= DIOC_LENGTH THEN
			nSmSend					:= SM_DIOC_SEND_END;
		END_IF

	SM_DIOC_SEND_END:
		(* Message is sent, give at least 1 bit pause *)
		nSmSend						:= SM_DIOC_SEND_START;

	SM_DIOC_SEND_TEST:;

	SM_DIOC_SEND_ERROR:;

	ELSE;

END_CASE

(* Log to ringbuffer *)
IF nTxBufferContainsItems >= 0 AND nTxBufferContainsItems <= DIOC_MAXPRIORITY THEN
Dioc_Register := F_DIOC_20_MESSAGE_IN(fbTxBuffer[nTxBufferContainsItems].OUT);
fbDioc_Ring_Tx(
	nPLC_Cycle	:= nPLC_Cycle,
	IN			:= Dioc_Register,
	WD			:= bTxRingBuffer_Write
	);
END_IF
END_ACTION

ACTION Startup:
;
END_ACTION

END_FUNCTION_BLOCK

// POUs/DIOC/_Internal/DIOC_HELPFUNCTIONS/FB_DIOC_FIFO
FUNCTION_BLOCK FB_DIOC_FIFO
VAR_INPUT
	IN		: A_DIOC_MESSAGE;	(* Value to be stored *)
	E 		: BOOL := TRUE;		(* Enable *)
	RST 	: BOOL;				(* Reset buffer *)
	fifo	: POINTER TO ARRAY[0..DIOC_RXTX_BUFFERSIZE] OF A_DIOC_MESSAGE;	(* pointer to first element of priority value buffer *)
END_VAR
VAR_OUTPUT
	OUT 	: A_DIOC_MESSAGE;	(* retrieved value *)
	EMPTY 	: BOOL := TRUE;		(* Buffer is empty *)
	FULL 	: BOOL;				(* Buffer full *)
END_VAR
VAR_IN_OUT
	RD 		: BOOL;				(* Read *)
	WD 		: BOOL;				(* Write *)
END_VAR
VAR
	pr 		: INT;				(* read pointer *)
	pw 		: INT;				(* Write pointer *)
END_VAR

IF RST THEN
	pw 						:= pr;
	FULL 					:= FALSE;
	EMPTY 					:= TRUE;
	OUT		 				:= 0;
ELSIF E THEN
	IF NOT EMPTY AND RD THEN
		OUT 				:= fifo^[pr];
		pr 					:= F_DIOC_INC2(pr,DIOC_RXTX_BUFFERSIZE);
		EMPTY 				:= pr = pw;
		FULL 				:= FALSE;
		RD					:= FALSE;			(* reset read request *)
	END_IF;
	IF NOT FULL AND WD THEN
		fifo^[pw]		 	:= IN;
		pw 					:= F_DIOC_INC2(pw,DIOC_RXTX_BUFFERSIZE);
		FULL 				:= pw = pr;
		EMPTY 				:= FALSE;
		WD					:= FALSE;			(* Reset write request *)
	END_IF;
END_IF;

END_FUNCTION_BLOCK

// POUs/DIOC/_Internal/DIOC_HELPFUNCTIONS/F_DIOC_INC2
FUNCTION F_DIOC_INC2 : INT
VAR_INPUT
	X : INT;
	N : INT;		(* Max value in loop *)
END_VAR



(*
version 1.2	23. feb. 2009
programmer 	kim
tested by	oscat

This is a increment function which increments the variable X by 1 and if N is reached, it begins with 0 instead of N again.
inc1(X,3) will generate 0,1,2,3,0,1,2,3,0,.....

*)

IF X >= N THEN
	F_DIOC_INC2 := 0;
ELSE
	F_DIOC_INC2 := X + 1;
END_IF;



(* revision history
hm	13. oct. 2008	rev 1.0
	original version

hm	22. oct. 2008	rev 1.1
	added statement to return value for compatibility reasons

hm	23. feb. 2009	rev 1.2
 	when inc1 is called with X >= N inc will continue with 0
*)

END_FUNCTION

// POUs/DIOC/_Internal/DIOC_HELPFUNCTIONS/FB_DIOC_RING
FUNCTION_BLOCK FB_DIOC_RING
VAR_INPUT
	nPLC_Cycle	: WORD;			(* Debugging *)
	IN		: ST_DIOC_REGISTER;	(* Value to be stored *)
	E 		: BOOL := TRUE;		(* Enable *)
	RST 	: BOOL;				(* Reset buffer *)
END_VAR
VAR_OUTPUT
	OUT 	: ST_DIOC_REGISTER;	(* last register *)
END_VAR
VAR_IN_OUT
	WD 		: BOOL;				(* Write *)
END_VAR
VAR
	ring	: ARRAY[0..DIOC_MAXRINGBUFFERSIZE] OF ST_DIOC_REGISTER;	(* local ringbuffer *)
	pw 		: INT;				(* Write pointer *)
	i: INT;
END_VAR

IF RST THEN
	pw 						:= 0;
	OUT.nRegister			:= 0;
	OUT.nValue				:= 0;
	FOR i := 0 TO	DIOC_MAXRINGBUFFERSIZE DO
		ring[i].nPLC_Cycle	:= 0;
		ring[i].nRegister	:= 0;
		ring[i].nValue		:= 0;
	END_FOR
	RST := FALSE;
ELSIF E AND wd THEN
	ring[pw].nPLC_Cycle		:= nPLC_Cycle;
	ring[pw].nRegister		:= in.nRegister;
	ring[pw].nValue			:= in.nValue;
	OUT 					:= ring[pw];
	pw 						:= F_DIOC_INC2(pw,DIOC_MAXRINGBUFFERSIZE);
	wd						:= FALSE;
END_IF;

END_FUNCTION_BLOCK

// POUs/DIOC/_Internal/DIOC/FB_DIOC_GEN
FUNCTION_BLOCK FB_DIOC_GEN
VAR_INPUT
	(* Data handshake interface *)
	in									: ST_DIOC_GEN_IN;
	in_Dioc_Status						: ST_DIOC_OUT;			(* Feedback dioc communication block *)
	Dioc_Register_IN					: ST_DIOC_REGISTER;		(* Message retrieved from buffer *)
	TYPE_ID								: DWORD;				(* Device identifier *)
END_VAR
VAR_OUTPUT
	(* Data feedback interface *)
	out									: ST_DIOC_GEN_OUT;
	nError								: E_DIOC_GEN_ERROR;
END_VAR
VAR_IN_OUT
	(*Dioc_Register_OUT					: A_DIOC_MESSAGE;*)
	RxBuffer							: ARRAY[0..DIOC_RXTX_BUFFERSIZE] OF A_DIOC_MESSAGE;	(* 1 message queue *)
	TxBuffer							: ARRAY[0..DIOC_MAXPRIORITY, 0..DIOC_RXTX_BUFFERSIZE] OF A_DIOC_MESSAGE;	(* 1 message queue / priority, HIGHEST: 0 = internal priority *)
	(* Fifo Buffer handlers *)
	fbRxBuffer							: FB_DIOC_FIFO;									(* 1 message queue *)
	fbTxBuffer							: ARRAY[0..DIOC_MAXPRIORITY] OF FB_DIOC_FIFO;	(* 1 message queue / priority *)
	(* Startup list *)
	arrstStartupParameter				: ARRAY[1..DIOC_NOOFSTARTUPPARAMETERS] OF ST_DIOC_REGISTER;
	(* Restarted ? *)
	bRestarted							: BOOL;

END_VAR
VAR CONSTANT
	DEVICE_CHARGE_TIME					: TIME 		:= T#2s;	(* Optional charge time *)
	SYNC_MESSAGE_REPEAT					: TIME 		:= T#5s;	(* Sync message repeat during cycle *)
	SYNC_MESSAGE_REPEAT_AT_STARTUP		: TIME 		:= T#500ms;	(* Sync message repeat at startup *)
	DIOC_LENGTH							: INT 		:= 21;		(* Dioc protocol length *)
	(*SYNC_MESSAGE						: DWORD		:= 2#0000_0000_000_1_1010_1010_1010_1111111_0;		(* Sync request = request type id *) (*not utilised anymore in newer firmware versions*)*)
	SYNC_MESSAGE_HIGH					: DWORD		:= 2#0000_0000_000_1_0101_0101_0101_0101010_0;		(* Sync request = request type id *)
END_VAR
VAR
(* TC3 attribute, will be ignored by TC2 *)
{attribute 'hide_all_locals'}
(* TC2 attribute, will be ignored by TC3 *)
{library private}
	(*
		RC State machine *)
	bHasBeenStarted						: BOOL;			(* Detect if the device has been fully started yet *)
	nSm									: E_SM_DIOC_DEVICE;
	nSmNextStep							: E_SM_DIOC_DEVICE;

	(* Previous state in *)
	stDeviceDataInPrevious				: ST_DIOC_GEN_IN;

	(* Ring buffer state machine *)
	ring								: ARRAY[0..DIOC_MAXRINGBUFFERSIZE] OF E_SM_DIOC_DEVICE;	(* local ringbuffer *)


	(*resend the enable bit*)
	_bSendEnable							: BOOL;

{library private}
	(*
		Timer sync message *)
	tSync								: TON;
	(*
		dioc communication *)
	stDiocRegister						: ST_DIOC_REGISTER;
	stDiocMessage						: A_DIOC_MESSAGE;
	nScrollPointerHW						: INT := -1;		(* Pointer if the device response >1 message *)
	nScrollPointerSW						: INT := -1;		(* Pointer if the device response >1 message *)
	nScrollPointerReg						: INT := -1;		(* Pointer if the device response >1 message *)
	nScrollPointerID						: INT := -1;		(* Pointer if the device response >1 message *)
	nScrollDateHW							: DWORD;			(* Date in dword format if the device response >1 message *)
	nScrollDateSW							: DWORD;			(* Date in dword format if the device response >1 message *)
	nScrollDateReg							: DWORD;			(* Date in dword format if the device response >1 message *)
	ptrScrollUniqueID					: POINTER TO ARRAY[1..24] OF BYTE;	(* Unique ID >1 message *)
	ptrScrollUniqueID_Hex				: POINTER TO ARRAY[1..2] OF BYTE;	(* Unique ID >1 message *)

	(*
		Sync message response, response is constructed at runtime, can depend on device *)
	dwSyncMessageResponse				: DWORD;

	(*
		device data IN, request to the device *)
	fpDeviceDataInNew					: R_TRIG;

	(*
		Startup list *)
	bStartup								: BOOL 		:= TRUE;
	nStartupValuePointer					: INT		:= 1;
	TonCyclicStartPar						: TON;
	nStartupValuePointerRepeat			: INT		:= 1;
	bDoubleStartPar						:BOOL;

	(* various *)
	i									: INT;
	byToggle							: DWORD;
	nPriority								: INT;		(* This value avoids copy paste errors, filled in by the program, see send action *)

	(* TEMP VARS *)
	nWriteRegister						: A_DIOC_DATA_TYPE;
	(* Buffer read / write *)
	bNoNewInputData						: BOOL;
	bRxBuffer_Read						: BOOL;
	bRxBuffer_Write						: BOOL;
	bTxBuffer_Read						: BOOL;
	bTxBuffer_Write						: BOOL;
	sR07_UniqueID						: STRING[24];				(* TEMP R7: Unique ID *)
	sR07_UniqueID_hex					: STRING[2];				(* TEMP R7: Unique ID *)

	(* Debug *)
	bRingWrite							: BOOL;
	fbRing								: FB_DIOC_RING2;

	(* Step / step *)
	bStepUnlocked						: BOOL;
	bSteplocked							: BOOL;
	bStepStepActive						: BOOL;
	bStepStep							: BOOL;
	fpStepStep							: R_TRIG;

	(* Increment and read error counter for testing purposes *)
	bSyncTest							: BOOL;
	bSyncTestOK							: BOOL;
	nSmSyncTest							: INT;
	nSyncCounter						: INT := 1;
	tSyncTest							: TON;

	(* Test timer to check if the device is not trying to restart*)
	tDeviceRestart : TON;


END_VAR

(*
	startup *)
IF bStartup THEN Startup(); END_IF

(*
	Toggle byte *)
byToggle		:= byToggle + 1;

(*
	Process new data from dioc *)
Receive();

(*
	RC State machine *)
(* Device deactivated? => reset state machine *)
IF NOT in_Dioc_Status.bDeviceReady 		THEN
	IF bHasBeenStarted					THEN
		(*bRestarted						:= TRUE;*)
		reset();
	END_IF
	nSmNextStep 	:= nSm				:= SM_DIOC_DEVICE_POWERUP_DEVICE;
END_IF

(* Step
	/ Step *)
fpStepStep(CLK:= bStepStep, Q=> );
bStepStep := FALSE;
bStepUnlocked 	:= nSmNextStep = nSm;
bSteplocked		:= NOT bStepUnlocked;
IF bSteplocked							THEN
	IF	bStepStepActive 				THEN
		IF fpStepStep.Q					THEN
			nSm							:= nSmNextStep;
		END_IF
	ELSE
		nSm								:= nSmNextStep;
	END_IF
END_IF

CASE nSm								OF

	SM_DIOC_DEVICE_POWERUP_DEVICE:				(* Power up device *)
		bHasBeenStarted					:= FALSE;
		tSync.PT						:= SYNC_MESSAGE_REPEAT_AT_STARTUP;
		IF in_Dioc_Status.bDeviceReady	THEN
			(* Reset the device statusses *)
			Reset();
			fbRing.RST 					:= TRUE;
			nSmNextStep					:= SM_DIOC_DEVICE_SEND_SYNC_REQUEST;
		END_IF

	SM_DIOC_DEVICE_SEND_SYNC_REQUEST:			(* sync message by master every 1 second until the device answers with the correct id *)
		IF tSync.Q	AND NOT fbTxBuffer[0].FULL AND bStepUnlocked THEN
			bTxBuffer_Write				:= TRUE;
			(* Store message in fifo queue *)
			fbTxBuffer[0](
				IN						:= SYNC_MESSAGE_HIGH,
				RD						:= bTxBuffer_Read,			(* Not functional *)
				WD						:= bTxBuffer_Write,
				fifo					:= ADR(TxBuffer[0, 0]));  	(* pointer to first element of the priority buffer 0 *)
			nSmNextStep					:= SM_DIOC_DEVICE_WAIT_FOR_TYPE_ID;
		END_IF

	SM_DIOC_DEVICE_WAIT_FOR_TYPE_ID:					(*Repeat sync message +  Message received ? Check the type id *)
		tSync.IN								 :=TRUE;
		IF tSync.Q	AND NOT fbTxBuffer[0].FULL AND bStepUnlocked THEN
				bTxBuffer_Write				:= TRUE;
				(* Store message in fifo queue *)
				fbTxBuffer[0](
					IN						:= SYNC_MESSAGE_HIGH,
					RD						:= bTxBuffer_Read,			(* Not functional *)
					WD						:= bTxBuffer_Write,
					fifo					:= ADR(TxBuffer[0, 0]));  	(* pointer to first element of the priority buffer 0 *)
			END_IF

		IF NOT in_Dioc_Status.bRxBufferEmpty	AND bStepUnlocked THEN

			bRxBuffer_Read				:= TRUE;
			fbRxBuffer(
				RD						:= bRxBuffer_Read,
				WD						:= bRxBuffer_Write,			(* Not functional *)
				fifo					:= ADR(RxBuffer));
			Dioc_Register_IN := F_DIOC_20_MESSAGE_IN(fbRxBuffer.OUT);
			(* Check the received message *)
			IF Dioc_Register_IN.nRegister = DIOC_R03_TYPE_ID AND Dioc_Register_IN.nValue = TYPE_ID	THEN
				nSmNextStep				:= SM_DIOC_DEVICE_SEND_SYNC_ACK;
			(*	tSync.PT				:= SYNC_MESSAGE_REPEAT;*)
			END_IF
		END_IF

	SM_DIOC_DEVICE_SEND_SYNC_ACK:					(* sync acknowledge by master *)
		(* Wait until the buffer is empty *)
		IF in_Dioc_Status.bTxBufferEmpty	AND bStepUnlocked THEN
			(* set auto send interval to 0 *)
			fbTxBuffer[0].IN := F_DIOC_20_MESSAGE_OUT(
				nRegister 	:= DIOC_R02_REGISTER_INTERVAL,		(* Request type ID *)
				nValue 		:= 0);
			(* Store message in fifo queue *)
			bTxBuffer_Write	:= TRUE;
			fbTxBuffer[0](
				RD							:= bTxBuffer_Read,
				WD							:= bTxBuffer_Write,
				fifo						:= ADR(TxBuffer[0, 0]));  (* pointer to first element of the priority buffer 0 *)
			(* set register request to Type ID *)
			fbTxBuffer[0].IN := F_DIOC_20_MESSAGE_OUT(
				nRegister 	:= DIOC_R01_REGISTER_REQUEST,		(* Request type ID *)
				nValue 		:= DIOC_R03_TYPE_ID);
			(* Store message in fifo queue *)
			bTxBuffer_Write	:= TRUE;
			fbTxBuffer[0](
				RD							:= bTxBuffer_Read,
				WD							:= bTxBuffer_Write,
				fifo						:= ADR(TxBuffer[0, 0]));  (* pointer to first element of the priority buffer 0 *)
			nStartupValuePointer			:= 1;
			nSmNextStep						:= SM_DIOC_DEVICE_DEVICE_ENABLE;
		END_IF

	SM_DIOC_DEVICE_DEVICE_ENABLE:					(* OPTIONAL Enable Device *)
		IF fbTxBuffer[0].empty AND	tSync.Q	AND bStepUnlocked THEN
			IF _bSendEnable THEN
				(* try to enable device*)
				(* set auto send interval to 0 *)
				fbTxBuffer[0].IN := F_DIOC_20_MESSAGE_OUT(
					nRegister 	:= DIOC_R11_DEVICE_ENABLE,		(* enable device *)
					nValue 		:= 1);
				(* Store message in fifo queue *)
				bTxBuffer_Write					:= TRUE;
				fbTxBuffer[0](
					RD							:= bTxBuffer_Read,
					WD							:= bTxBuffer_Write,
					fifo						:= ADR(TxBuffer[0, 0]));  (* pointer to first element of the priority buffer 0 *)
					_bSendEnable := FALSE;
			ELSE
				(* try to enable device*)
				(* set auto send interval to 0 *)
				fbTxBuffer[0].IN := F_DIOC_20_MESSAGE_OUT(
					nRegister := DIOC_R01_REGISTER_REQUEST,
					nValue := DIOC_R11_DEVICE_ENABLE);
				(* Store message in fifo queue *)
				bTxBuffer_Write					:= TRUE;
				fbTxBuffer[0](
					RD							:= bTxBuffer_Read,
					WD							:= bTxBuffer_Write,
					fifo						:= ADR(TxBuffer[0, 0]));  (* pointer to first element of the priority buffer 0 *)
					_bSendEnable := TRUE;
			END_IF
		END_IF

		IF NOT in_Dioc_Status.bRxBufferEmpty	AND bStepUnlocked THEN

			bRxBuffer_Read				:= TRUE;
			fbRxBuffer(
				RD						:= bRxBuffer_Read,
				WD						:= bRxBuffer_Write,			(* Not functional *)
				fifo					:= ADR(RxBuffer));
			Dioc_Register_IN := F_DIOC_20_MESSAGE_IN(fbRxBuffer.OUT);
			(* Check the received message *)
			IF Dioc_Register_IN.nRegister = DIOC_R11_DEVICE_ENABLE AND Dioc_Register_IN.nValue.0 = TRUE THEN (* this means the device is active*)

				nSmNextStep				:= SM_DIOC_DEVICE_SEND_STARTUP_VALUES;
				tSync.PT				:= SYNC_MESSAGE_REPEAT;
			END_IF
		END_IF

	SM_DIOC_DEVICE_SEND_STARTUP_VALUES:			(* OPTIONAL Send optional startup values *)
		(* Send startup values, 1 every cycle, until startup list is processed *)
		IF  fbTxBuffer[0].empty	AND bStepUnlocked THEN
			(* Shift all parameters to priority 0 (HIGHEST) *)
			IF arrstStartupParameter[nStartupValuePointer].nRegister <> 0 AND arrstStartupParameter[nStartupValuePointer].nRegister <> DIOC_INVALID_REGISTER THEN
				fbTxBuffer[0].IN := F_DIOC_20_MESSAGE_OUT(
					nRegister 	:= arrstStartupParameter[nStartupValuePointer].nRegister,		(* Request type ID *)
					nValue 		:= arrstStartupParameter[nStartupValuePointer].nValue);
				(* Store message in fifo queue *)
				bTxBuffer_Write				:= TRUE;
				fbTxBuffer[0](
					RD						:= bTxBuffer_Read,
					WD						:= bTxBuffer_Write,
					fifo					:= ADR(TxBuffer[0, 0]));  (* pointer to first element of the priority buffer 0 *)
			END_IF;
			nStartupValuePointer		:= nStartupValuePointer + 1;
			IF nStartupValuePointer > DIOC_NOOFSTARTUPPARAMETERS THEN
                nSmNextStep                                                                   := SM_DIOC_DEVICE_STARTUP_VALUES_SENT;
			ELSIF arrstStartupParameter[nStartupValuePointer].nRegister = DIOC_INVALID_REGISTER THEN
                nSmNextStep                                                                   := SM_DIOC_DEVICE_STARTUP_VALUES_SENT;
			END_IF

		END_IF

	SM_DIOC_DEVICE_STARTUP_VALUES_SENT:			(* OPTIONAL Send optional startup values *)
		(* Wait until the send buffer is empty *)
		IF fbTxBuffer[0].empty				AND bStepUnlocked THEN
			nSmNextStep 					:= SM_DIOC_DEVICE_DEVICE_ENABLED;
			bRestarted						:= TRUE;
		END_IF


	SM_DIOC_DEVICE_DEVICE_ENABLED:					(* OPTIONAL Enable Device *)
		(* Wait until the buffer is empty *)
		IF fbTxBuffer[0].empty				AND bStepUnlocked THEN
			IF bRestarted					THEN
				nSmNextStep 				:= SM_DIOC_DEVICE_RESTART;
			ELSE
				nSmNextStep 				:= SM_DIOC_DEVICE_ACTIVE;
			END_IF
		END_IF

	SM_DIOC_DEVICE_RESTART:					(* Wait until the device parameters have been re-written after restart *)
		Restart();
		nSmNextStep 						:= SM_DIOC_DEVICE_ACTIVE;

	SM_DIOC_DEVICE_ACTIVE:					(* device is active *)
		bHasBeenStarted						:= TRUE;	(* Remember it has been started *)
		(* Increment and read error counter for testing purposes *)
		tSyncTest(IN:= (nSmSyncTest=2) OR (nSmSyncTest=4), PT:= t#250ms, Q=> , ET=> );
		IF	bSyncTest	AND nSmSyncTest = 0 THEN
			nSmSyncTest := nSmSyncTest + 1;
			in.bR08_Message_Error_Counter_WRITE		:= TRUE;
			bSyncTestOK								:= TRUE;
			in.nR08_MessageErrorCounter				:= INT_TO_UINT(nSyncCounter);
		ELSIF NOT bSyncTest			THEN
			nSmSyncTest := 0;
		END_IF
		(* Test case *)
		CASE nSmSyncTest		OF

			0:;

			1:
				in.bR08_Message_Error_Counter_READ	:= TRUE;
				out.nR08_MessageErrorCounter 		:= 65535;
				nSmSyncTest 						:= nSmSyncTest + 1;

			2:
				IF tSyncTest.Q						THEN
					nSmSyncTest 					:= nSmSyncTest + 1;
				END_IF

			3:
				IF out.nR08_MessageErrorCounter < 65535 	THEN
					IF NOT (out.nR08_MessageErrorCounter = INT_TO_UINT(nSyncCounter))		THEN
						bSyncTestOK					:= FALSE;
					ELSE
						bSyncTestOK					:= TRUE;
						in.bR08_Message_Error_Counter_WRITE	:= TRUE;
						nSyncCounter				:= nSyncCounter + 1;
						in.nR08_MessageErrorCounter	:= INT_TO_UINT(nSyncCounter);
						nSmSyncTest 				:= nSmSyncTest + 1;
					END_IF
				END_IF

			4:
				IF tSyncTest.Q						THEN
					nSmSyncTest 					:= 1;
				END_IF

			ELSE;

		END_CASE

	SM_DIOC_DEVICE_END:;

	SM_DIOC_DEVICE_TEST:;

	SM_DIOC_DEVICE_ERROR:;

	ELSE;

END_CASE

(* Device is active *)
out.bDeviceActive := nSmNextStep = SM_DIOC_DEVICE_ACTIVE;

(*	External Dioc request processing, with priority handling *)
Send();

fbRing(
	IN			:= nSm,
	AUTO		:= TRUE,
	WD			:= bRingWrite,
	ring		=>
	);
MEMCPY(ADR(ring), ADR(fbRing.OUT), SIZEOF(ring));

(*
	Timers *)

tSync(IN := NOT tSync.Q AND NOT (nSm = SM_DIOC_DEVICE_SEND_STARTUP_VALUES), PT:= , Q=> , ET=> );

(* auto repeated sync *)
IF tSync.Q	AND NOT fbTxBuffer[0].FULL 	THEN
	(* Trigger sync message *)
	in.bR00_SyncMessage					:= TRUE;
END_IF

(* Check if the DIOC device is not trying to restart *)

	(* timer is true when no info has been received to register 3 the last minute*)
	tDeviceRestart(IN:= ((nSm = SM_DIOC_DEVICE_ACTIVE) AND Dioc_Register_IN.nRegister = 3), PT:= t#1m);

	(* If data is received multiple times per minute on register 3,the device is probably trying to restart the communication*)
	IF tDeviceRestart.q THEN
		nSmNextStep 				:= SM_DIOC_DEVICE_POWERUP_DEVICE;
	END_IF

(* Cyclic repeat of Startup Vars *)
TonCyclicStartPar(IN:= (NOT TonCyclicStartPar.q) AND (nSm = SM_DIOC_DEVICE_ACTIVE), PT:= T#5s, Q=> , ET=> );
IF (TonCyclicStartPar.q) OR bDoubleStartPar THEN
	nStartupValuePointerRepeat := nStartupValuePointerRepeat +1;
	IF (arrstStartupParameter[nStartupValuePointerRepeat].nRegister = 0) THEN
		nStartupValuePointerRepeat := 1;
	END_IF
	in.bRxx_StartPar := TRUE;
	IF arrstStartupParameter[nStartupValuePointerRepeat].nRegister = 2 THEN
		bDoubleStartPar := TRUE;
	ELSE
		bDoubleStartPar := FALSE;
	END_IF;
END_IF


(*
	First loop finished *)
bStartup 					:= FALSE;

ACTION Receive:
(* !!! ONLY ACTIVE WHEN THE DEVICE IS ACTIVE !!! *)

(*New dioc data received and the device is active *)
IF in_Dioc_Status.bRxBufferEmpty	OR NOT out.bDeviceActive THEN
	out.nRxx_Received 					:= -1;
	out.bRxx_Received 					:= FALSE;
	RETURN;
END_IF

(*New data received *)
out.nRxx_Received 						:= Dioc_Register_IN.nRegister;
out.bRxx_Received 						:= TRUE;

(*Process new data *)
CASE Dioc_Register_IN.nRegister			OF

	DIOC_R03_TYPE_ID:					(*3*)
		out.nR03_TypeID					:= DWORD_TO_INT(Dioc_Register_IN.nValue);

	DIOC_R04_VERSION_HW:					(*4*)
		IF Dioc_Register_IN.nValue = 170	THEN 	(* 170d, AAh *)
			nScrollPointerHW 			:= 0;
			nScrollDateHW				:= 0;
			in.bR04_Request_HW_Version	:= TRUE;
		ELSIF nScrollPointerHW >= 0 		THEN
			nScrollDateHW 				:= nScrollDateHW + (Dioc_Register_IN.nValue - 48) * REAL_TO_DWORD(EXPT(10, 5-nScrollpointerHW));
			IF nScrollPointerHW >= 5 		THEN
				out.dtR04_VersionHW		:= F_DIOC_TO_DATE(nScrollDateHW);
				nScrollPointerHW 			:= -1;
			ELSE
				in.bR04_Request_HW_Version	:= TRUE;
				nScrollPointerHW 			:= nScrollPointerHW + 1;
			END_IF
		ELSE
			in.bR04_Request_HW_Version	:= TRUE;	(* Keep scrolling looking for start char *)
		END_IF

	DIOC_R05_VERSION_SW:					(*5*)
		IF Dioc_Register_IN.nValue = 170	THEN 	(* 170d, AAh *)
			nScrollPointerSW 			:= 0;
			nScrollDateSW				:= 0;
			in.bR05_Request_SW_Version	:= TRUE;
		ELSIF nScrollPointerSW >= 0 		THEN
			nScrollDateSW 				:= nScrollDateSW + (Dioc_Register_IN.nValue - 48) * REAL_TO_DWORD(EXPT(10, 5-nScrollpointerSW));
			IF nScrollPointerSW >= 5 		THEN
				out.dtR05_VersionSW		:= F_DIOC_TO_DATE(nScrollDateSW);
				nScrollPointerSW 			:= -1;
			ELSE
				in.bR05_Request_SW_Version	:= TRUE;
				nScrollPointerSW 			:= nScrollPointerSW + 1;
			END_IF
		ELSE
			in.bR05_Request_SW_Version	:= TRUE;	(* Keep scrolling looking for start char *)
		END_IF

	DIOC_R06_VERSION_REGISTERS:				(*6*)
		IF Dioc_Register_IN.nValue = 170	THEN 	(* 170d, AAh *)
			nScrollPointerREG 			:= 0;
			nScrollDateREG				:= 0;
			in.bR06_Request_Register_Version	:= TRUE;
		ELSIF nScrollPointerREG >= 0 		THEN
			nScrollDateREG 				:= nScrollDateREG + (Dioc_Register_IN.nValue - 48) * REAL_TO_DWORD(EXPT(10, 5-nScrollpointerREG));
			IF nScrollPointerREG >= 5 		THEN
				out.dtR06_VersionREG	:= F_DIOC_TO_DATE(nScrollDateREG);
				nScrollPointerREG 			:= -1;
			ELSE
				in.bR06_Request_Register_Version	:= TRUE;
				nScrollPointerREG 			:= nScrollPointerREG + 1;
			END_IF
		ELSE
			in.bR06_Request_Register_Version	:= TRUE;	(* Keep scrolling looking for start char *)
		END_IF

	DIOC_R07_UNIQUE_ID:						(*7*)
		ptrScrollUniqueID				:= ADR(sR07_UniqueID);
		ptrScrollUniqueID_Hex			:= ADR(sR07_UniqueID_hex);
		IF Dioc_Register_IN.nValue = 170	THEN 	(* 170d, AAh *)
			out.sR07_UniqueID			:= '';
			nScrollPointerID 				:= 1;
			sR07_UniqueID				:= '';		(* Internal *)
			in.bR07_Request_Unique_ID	:= TRUE;	(* Keep scrolling looking for start char *)
		ELSIF nScrollPointerID >= 0		THEN
			sR07_UniqueID_hex := DWORD_TO_HEXSTR(Dioc_Register_IN.nValue, 2, FALSE);
			ptrScrollUniqueID^[nScrollPointerID] := ptrScrollUniqueID_Hex^[1];
			ptrScrollUniqueID^[nScrollPointerID + 1] := ptrScrollUniqueID_Hex^[2];
			IF nScrollPointerID >= 23 	THEN
				out.sR07_UniqueID		:= sR07_UniqueID;
				nScrollPointerID 			:= -1;
			ELSE
				in.bR07_Request_Unique_ID	:= TRUE;	(* Keep scrolling looking for start char *)
				nScrollPointerID 			:= nScrollPointerID + 2;
			END_IF
		ELSE
			in.bR07_Request_Unique_ID	:= TRUE;	(* Keep scrolling looking for start char *)
		END_IF

	DIOC_R08_MESSAGE_ERROR_COUNTER:			(*8*)
		out.nR08_MessageErrorCounter			:= DWORD_TO_UINT(Dioc_Register_IN.nValue);

	DIOC_R09_VOLTAGE_LEVEL_A:				(*9*)
		out.nR09_DiocVoltageA				:= F_SCALE_FROM_DIOC(Dioc_Register_IN.nValue, 0, 511, 0, 51.1, 0);

	DIOC_R10_VOLTAGE_LEVEL_B:				(*10*)
		out.nR10_DiocVoltageB				:= F_SCALE_FROM_DIOC(Dioc_Register_IN.nValue, 0, 511, 0, 51.1, 0);

	DIOC_R11_DEVICE_ENABLE:					(*11*)
		out.bR11_DeviceEnabled				:= Dioc_Register_IN.nValue.0;

	DIOC_R12_CPU_TEMPERATURE:				(*12*)
		out.nR12_CpuTemperature 				:= F_SCALE_FROM_DIOC(Dioc_Register_IN.nValue, 0, 4095, -20, 120, -20);

	DIOC_R13_ErrorRegisterAdress:			(*13*)
		out.nR13_ErrorRegisterAdress			:= DWORD_TO_UINT(Dioc_Register_IN.nValue);
		IF	gv_dioc_sSystemTimeString = '' 	THEN
			out.sR13_DtLastError				:= UDINT_TO_STRING(byToggle);
		ELSE
			out.sR13_DtLastError				:= gv_dioc_sSystemTimeString;
		END_IF

	TP10_TRANSMIT_DELAY:					(*84*)
		out.nR84_TransmitDelay 				:= F_SCALE_FROM_DIOC(Dioc_Register_IN.nValue, 0, 100, 0, 100, 0);

	TP10_SYNC_MESSAGE_HIGH	:;


	ELSE;

END_CASE
END_ACTION

ACTION Reset:
(*  FEEDBACK
	Reset all output statusses *)
out.bR11_DeviceEnabled				:= FALSE;						(* R11: Device Enable *)

(* RC register feedback values *)
out.nR03_TypeID						:= 0;							(* R3: Type ID *)
out.nR08_MessageErrorCounter		:= 0;							(* R8: Message Err. Counter *)
out.dtR04_VersionHW					:= D#1970-01-01;				(* R4: Version HW, 7 scrolls *)
out.dtR05_VersionSW					:= D#1970-01-01;				(* R5: Version SW, 7 scrolls *)
out.dtR06_VersionREG				:= D#1970-01-01;				(* R6: Version Registers, 7 scrolls *)
out.sR07_UniqueID					:= '';							(* R7: Unique ID *)
out.nR09_DiocVoltageA				:= -3.402823E38; 				(* R9: Read DIOCA voltage level (x10) *)
out.nR10_DiocVoltageB				:= -3.402823E38; 				(* R10: Read DIOCA voltage level (x10) *)
out.nR12_CpuTemperature				:= -3.402823E38; 				(* R12: CPU Temperature *)
out.nR84_TransmitDelay				:= -3.402823E38;				(* R84: 'transmit delay (timeshift PLC<-> device) *)

(* Internal values *)
nScrollPointerHW := 0;
nScrollPointerSW := 0;
nScrollPointerReg := 0;
nScrollPointerID := 0;
END_ACTION

ACTION Restart:
(*
	Possible actions after restart of the dioc *)
;
END_ACTION

ACTION Send:
(* !!! ONLY ACTIVE WHEN THE DEVICE IS ACTIVE !!! *)

(*
	is the device active *)
IF nSm <> SM_DIOC_DEVICE_ACTIVE THEN
	RETURN;
END_IF

(*
	New dioc input data received ? *)
bNoNewInputData := MEMCMP(ADR(stDeviceDataInPrevious), ADR(in), SIZEOF(stDeviceDataInPrevious)) = 0;
IF bNoNewInputData THEN RETURN; END_IF;

(*
	Handle register handling in the order of priority *)
(* PRIORITY 00: internal commands (eg at startup) *)
(* Test message, highest priority, always send a sync message first *)
nPriority := 0;

IF	in.bRxx_SendMessage				THEN
	fbTxBuffer[nPriority](
		IN							:= F_DIOC_20_MESSAGE_OUT(nRegister := in.byRxx_SendMessageRegister, nValue := in.dwRxx_SendMessageData),
		RD							:= bTxBuffer_Read,	(* Not functional *)
		WD							:= in.bRxx_SendMessage,
		fifo						:= ADR(TxBuffer[nPriority, 0]));

END_IF

IF in.bR00_SyncMessage THEN	(* external / internal sync request *)
	fbTxBuffer[nPriority](
		IN							:=  F_DIOC_20_MESSAGE_OUT(nRegister := 85, nValue := 2730),
		RD							:= bTxBuffer_Read,	(* Not functional *)
		WD							:= in.bR00_SyncMessage,
		fifo						:= ADR(TxBuffer[nPriority, 0]));  (* pointer to first element of the priority buffer 0 *)
END_IF
(* PRIORITY 01 *)
nPriority := 1;

(*startup list*)
IF in.bRxx_StartPar THEN
	fbTxBuffer[nPriority](
		IN							:= F_DIOC_20_MESSAGE_OUT(nRegister := arrstStartupParameter[nStartupValuePointerRepeat].nRegister, nValue := arrstStartupParameter[nStartupValuePointerRepeat].nValue),
		RD							:= bTxBuffer_Read,			(* Not functional *)
		WD							:= in.bRxx_StartPar,
		fifo						:= ADR(TxBuffer[nPriority, 0]));	(* Send the register *)
END_IF

(* Transmit delay *)
IF	in.bR84_TransmitDelay_WRITE		THEN
	fbTxBuffer[nPriority](
		IN							:= F_DIOC_20_MESSAGE_OUT(nRegister := TP10_TRANSMIT_DELAY, nValue := in.dwR84_TransmitDelay),
		RD							:= bTxBuffer_Read,	(* Not functional *)
		WD							:= in.bR84_TransmitDelay_WRITE,
		fifo						:= ADR(TxBuffer[nPriority, 0]));
END_IF

IF	in.bR84_TransmitDelay_READ		THEN
	out.nR84_TransmitDelay			:= -1;
	fbTxBuffer[nPriority](
		IN							:= F_DIOC_20_MESSAGE_OUT(nRegister := DIOC_R01_REGISTER_REQUEST, nValue := TP10_TRANSMIT_DELAY),
		RD							:= bTxBuffer_Read,	(* Not functional *)
		WD							:= in.bR84_TransmitDelay_READ,
		fifo						:= ADR(TxBuffer[nPriority, 0]));
END_IF


(* Register request, send interval *)
IF	in.bR01_RegisterRequestAutoSend	THEN
	bTxBuffer_Write					:= TRUE;
	fbTxBuffer[nPriority](
		IN							:= F_DIOC_20_MESSAGE_OUT(nRegister := DIOC_R02_REGISTER_INTERVAL, nValue := in.dwR02_MessageAutoSendInterval),
		RD							:= bTxBuffer_Read,			(* Not functional *)
		WD							:= bTxBuffer_Write,
		fifo						:= ADR(TxBuffer[nPriority, 0]));	(* Send the register *)
END_IF

IF	in.bR01_RegisterRequest			THEN
	fbTxBuffer[nPriority](
		IN							:= F_DIOC_20_MESSAGE_OUT(nRegister := DIOC_R01_REGISTER_REQUEST, nValue := in.dwR01_MessageRegister),
		RD							:= bTxBuffer_Read,			(* Not functional *)
		WD							:= in.bR01_RegisterRequest,
		fifo						:= ADR(TxBuffer[nPriority, 0]));
END_IF

IF	in.bR01_RegisterRequestAutoSend	THEN
	fbTxBuffer[nPriority](
		IN							:= F_DIOC_20_MESSAGE_OUT(nRegister := DIOC_R01_REGISTER_REQUEST, nValue := in.dwR01_MessageRegister),
		RD							:= bTxBuffer_Read,			(* Not functional *)
		WD							:= in.bR01_RegisterRequestAutoSend,
		fifo						:= ADR(TxBuffer[nPriority, 0]));
END_IF

(* PRIORITY 02 *)
nPriority := 2;

(* PRIORITY 03 *)
nPriority := 3;

(* PRIORITY 04 *)
nPriority := 4;

(* PRIORITY 05 *)
nPriority := 5;

(* PRIORITY 06 *)
nPriority := 6;
IF in.bR08_Message_Error_Counter_WRITE	THEN
	bTxBuffer_Write					:= TRUE;
	fbTxBuffer[nPriority](
		IN							:= F_DIOC_20_MESSAGE_OUT(nRegister := DIOC_R08_MESSAGE_ERROR_COUNTER, nValue := in.nR08_MessageErrorCounter),
		RD							:= bTxBuffer_Read,			(* Not functional *)
		WD							:= bTxBuffer_Write,
		fifo						:= ADR(TxBuffer[nPriority, 0]));
	out.nR08_MessageErrorCounter	:= 65535;
	fbTxBuffer[nPriority](
		IN							:= F_DIOC_20_MESSAGE_OUT(nRegister := DIOC_R01_REGISTER_REQUEST, nValue := DIOC_R08_MESSAGE_ERROR_COUNTER),
		RD							:= bTxBuffer_Read,			(* Not functional *)
		WD							:= in.bR08_Message_Error_Counter_WRITE,
		fifo						:= ADR(TxBuffer[nPriority, 0]));
END_IF

(* PRIORITY 07 *)
nPriority := 7;

(* PRIORITY 08 *)
nPriority := 8;
(* Request TYPE ID *)
IF	in.bR03_Request_Type_ID			THEN
	out.nR03_TypeID					:= -1;
	fbTxBuffer[nPriority](
		IN							:= F_DIOC_20_MESSAGE_OUT(nRegister := DIOC_R01_REGISTER_REQUEST, nValue := DIOC_R03_TYPE_ID),
		RD							:= bTxBuffer_Read,			(* Not functional *)
		WD							:= in.bR03_Request_Type_ID,
		fifo						:= ADR(TxBuffer[nPriority, 0]));
END_IF

IF	in.bR04_Request_HW_Version		THEN
	fbTxBuffer[nPriority](
		IN							:= F_DIOC_20_MESSAGE_OUT(nRegister := DIOC_R01_REGISTER_REQUEST, nValue := DIOC_R04_VERSION_HW),
		RD							:= bTxBuffer_Read,			(* Not functional *)
		WD							:= in.bR04_Request_HW_Version,
		fifo						:= ADR(TxBuffer[nPriority, 0]));
END_IF

IF	in.bR05_Request_SW_Version		THEN
	fbTxBuffer[nPriority](
		IN							:= F_DIOC_20_MESSAGE_OUT(nRegister := DIOC_R01_REGISTER_REQUEST, nValue := DIOC_R05_VERSION_SW),
		RD							:= bTxBuffer_Read,			(* Not functional *)
		WD							:= in.bR05_Request_SW_Version,
		fifo						:= ADR(TxBuffer[nPriority, 0]));
END_IF

IF	in.bR06_Request_Register_Version	THEN
	fbTxBuffer[nPriority](
		IN							:= F_DIOC_20_MESSAGE_OUT(nRegister := DIOC_R01_REGISTER_REQUEST, nValue := DIOC_R06_VERSION_REGISTERS),
		RD							:= bTxBuffer_Read,			(* Not functional *)
		WD							:= in.bR06_Request_Register_Version,
		fifo						:= ADR(TxBuffer[nPriority, 0]));
END_IF

IF	in.bR07_Request_Unique_ID	THEN
	out.sR07_UniqueID				:= '';
	fbTxBuffer[nPriority](
		IN							:= F_DIOC_20_MESSAGE_OUT(nRegister := DIOC_R01_REGISTER_REQUEST, nValue := DIOC_R07_UNIQUE_ID),
		RD							:= bTxBuffer_Read,			(* Not functional *)
		WD							:= in.bR07_Request_Unique_ID,
		fifo						:= ADR(TxBuffer[nPriority, 0]));
END_IF

IF in.bR08_Message_Error_Counter_READ	THEN
	out.nR08_MessageErrorCounter	:= 65535;
	fbTxBuffer[nPriority](
		IN							:= F_DIOC_20_MESSAGE_OUT(nRegister := DIOC_R01_REGISTER_REQUEST, nValue := DIOC_R08_MESSAGE_ERROR_COUNTER),
		RD							:= bTxBuffer_Read,			(* Not functional *)
		WD							:= in.bR08_Message_Error_Counter_READ,
		fifo						:= ADR(TxBuffer[nPriority, 0]));
END_IF

IF in.bR09_Read_DiocA_Voltage_Level	THEN
	out.nR09_DiocVoltageA			:= -1;
	fbTxBuffer[nPriority](
		IN							:= F_DIOC_20_MESSAGE_OUT(nRegister := DIOC_R01_REGISTER_REQUEST, nValue := DIOC_R09_VOLTAGE_LEVEL_A),
		RD							:= bTxBuffer_Read,			(* Not functional *)
		WD							:= in.bR09_Read_DiocA_Voltage_Level,
		fifo						:= ADR(TxBuffer[nPriority, 0]));
END_IF

IF in.bR10_Read_DiocB_Voltage_Level	THEN
	out.nR10_DiocVoltageB			:= -1;
	fbTxBuffer[nPriority](
		IN							:= F_DIOC_20_MESSAGE_OUT(nRegister := DIOC_R01_REGISTER_REQUEST, nValue := DIOC_R10_VOLTAGE_LEVEL_B),
		RD							:= bTxBuffer_Read,			(* Not functional *)
		WD							:= in.bR10_Read_DiocB_Voltage_Level,
		fifo						:= ADR(TxBuffer[nPriority, 0]));
END_IF

IF in.bR11_Enable_Device_READ		THEN
	out.bR11_DeviceEnabled			:= FALSE;
	fbTxBuffer[nPriority](
		IN							:= F_DIOC_20_MESSAGE_OUT(nRegister := DIOC_R01_REGISTER_REQUEST, nValue := DIOC_R11_DEVICE_ENABLE),
		RD							:= bTxBuffer_Read,			(* Not functional *)
		WD							:= in.bR11_Enable_Device_READ,
		fifo						:= ADR(TxBuffer[nPriority, 0]));
END_IF

IF in.bR11_Enable_Device			THEN
	bTxBuffer_Write					:= TRUE;
	fbTxBuffer[nPriority](
		IN							:= F_DIOC_20_MESSAGE_OUT(nRegister := DIOC_R11_DEVICE_ENABLE, nValue := 1),
		RD							:= bTxBuffer_Read,			(* Not functional *)
		WD							:= bTxBuffer_Write,
		fifo						:= ADR(TxBuffer[nPriority, 0]));
	out.bR11_DeviceEnabled			:= FALSE;
	fbTxBuffer[nPriority](
		IN							:= F_DIOC_20_MESSAGE_OUT(nRegister := DIOC_R01_REGISTER_REQUEST, nValue := DIOC_R11_DEVICE_ENABLE),
		RD							:= bTxBuffer_Read,			(* Not functional *)
		WD							:= in.bR11_Enable_Device,
		fifo						:= ADR(TxBuffer[nPriority, 0]));
END_IF

IF in.bR11_Disable_Device			THEN
	bTxBuffer_Write					:= TRUE;
	fbTxBuffer[nPriority](
		IN							:= F_DIOC_20_MESSAGE_OUT(nRegister := DIOC_R11_DEVICE_ENABLE, nValue := 0),
		RD							:= bTxBuffer_Read,			(* Not functional *)
		WD							:= bTxBuffer_Write,
		fifo						:= ADR(TxBuffer[nPriority, 0]));
	out.bR11_DeviceEnabled			:= TRUE;
	fbTxBuffer[nPriority](
		IN							:= F_DIOC_20_MESSAGE_OUT(nRegister := DIOC_R01_REGISTER_REQUEST, nValue := DIOC_R11_DEVICE_ENABLE),
		RD							:= bTxBuffer_Read,			(* Not functional *)
		WD							:= in.bR11_Disable_Device,
		fifo						:= ADR(TxBuffer[nPriority, 0]));
END_IF

IF in.bR12_CPU_Temperature			THEN
	out.nR12_CpuTemperature			:= -1;
	fbTxBuffer[nPriority](
		IN							:= F_DIOC_20_MESSAGE_OUT(nRegister := DIOC_R01_REGISTER_REQUEST, nValue := DIOC_R12_CPU_TEMPERATURE),
		RD							:= bTxBuffer_Read,			(* Not functional *)
		WD							:= in.bR12_CPU_Temperature,
		fifo						:= ADR(TxBuffer[nPriority, 0]));
END_IF
END_ACTION

ACTION Startup:
;
END_ACTION

END_FUNCTION_BLOCK

// POUs/DIOC/_Internal/DIOC_HELPFUNCTIONS/FB_DIOC_RING2
FUNCTION_BLOCK FB_DIOC_RING2
VAR_INPUT
	IN		: INT;	(* Value to be stored *)
	AUTO	: BOOL;
	E 		: BOOL := TRUE;		(* Enable *)
	RST 	: BOOL;				(* Reset buffer *)
END_VAR
VAR_OUTPUT
	OUT 	: INT;	(* last register *)
	ring	: ARRAY[0..MAXRINGBUFFERSIZE] OF INT;	(* local ringbuffer *)
END_VAR
VAR_IN_OUT
	WD 		: BOOL;				(* Write *)
END_VAR
VAR CONSTANT
	MAXRINGBUFFERSIZE 		: INT := 20;
END_VAR
VAR
	WD_AUTO 				: BOOL;				(* Write *)
	in_previous				: INT;
	pw 						: INT;				(* Write pointer *)
	i: INT;
END_VAR

IF AUTO						THEN
	IF in <> in_previous	THEN
		wd_auto 			:= TRUE;
		in_previous 		:= in;
	END_IF
END_IF

IF RST THEN
	pw 						:= 0;
	OUT						:= 0;
	FOR i := 0 TO MAXRINGBUFFERSIZE	DO
		ring[i] := 0;
	END_FOR
	RST := FALSE;
ELSIF E AND (wd OR WD_AUTO) THEN
	ring[pw]				:= in;
	OUT 					:= ring[pw];
	pw 						:= F_DIOC_INC2(pw,MAXRINGBUFFERSIZE);
END_IF;

wd							:= FALSE;
WD_AUTO						:= FALSE;

END_FUNCTION_BLOCK

// POUs/DIOC/_Internal/DIOC_HELPFUNCTIONS/F_DIOC_TO_DATE
(*
	Converts a dioc date stream to PLC DATE Type *)
FUNCTION F_DIOC_TO_DATE : DATE
VAR_INPUT
	nDiocDate			: DWORD;
END_VAR
VAR
	TimeStr				: TIMESTRUCT;
END_VAR

Timestr.wDay			:= DWORD_TO_WORD(nDiocDate/10000 MOD 100);
Timestr.wMonth			:= DWORD_TO_WORD(nDiocDate/100 MOD 100);
Timestr.wYear			:= DWORD_TO_WORD(nDiocDate MOD 100) + 2000;
F_DIOC_TO_DATE			:= DT_TO_DATE(SYSTEMTIME_TO_DT(Timestr));

END_FUNCTION

// POUs/DIOC/_Internal/DIOC_HELPFUNCTIONS/F_SCALE_FROM_DIOC
FUNCTION F_SCALE_FROM_DIOC : REAL
VAR_INPUT
	nValue				: A_DIOC_DATA_TYPE;
	nRAWMin				: REAL;
	nRAWMax				: REAL;
	nSCALEDMin			: REAL;
	nSCALEDMax			: REAL;
	nSCALEDOffset		: REAL;
END_VAR
VAR
END_VAR

F_SCALE_FROM_DIOC := nSCALEDOffset + DWORD_TO_REAL(nValue) * (nSCALEDMax - nSCALEDMin) / (nRAWMax - nRAWMin);

END_FUNCTION

// POUs/DIOC/_Internal/DIOC_HELPFUNCTIONS/F_SCALE_FROM_DIOC_FO
FUNCTION F_SCALE_FROM_DIOC_FO : REAL
VAR_INPUT
	wX: DWORD;
	xGrens :REAL;
	yGrens : REAL;
	xLin: REAL;
END_VAR
VAR
	x : REAL;
END_VAR

x := DWORD_TO_REAL(wX);
IF x < xLin THEN
	F_SCALE_FROM_DIOC_FO := x;
ELSE
	F_SCALE_FROM_DIOC_FO := xLin + MAX(0,(ygrens-xLin)*(1-EXPT(2.72,-(x-1200)/(xGrens/4))));
END_IF

END_FUNCTION

// POUs/DIOC/_Internal/DIOC_HELPFUNCTIONS/F_SCALE_FROM_REAL
FUNCTION F_SCALE_FROM_REAL : REAL
VAR_INPUT
	nValue				: REAL;
	nRAWMin				: REAL;
	nRAWMax				: REAL;
	nSCALEDMin			: REAL;
	nSCALEDMax			: REAL;
	nSCALEDOffset		: REAL;
END_VAR
VAR
END_VAR

F_SCALE_FROM_REAL := nSCALEDOffset + nValue * (nSCALEDMax - nSCALEDMin) / (nRAWMax - nRAWMin);

END_FUNCTION

// POUs/DIOC/_Internal/DIOC_HELPFUNCTIONS/F_SCALE_TO_DIOC
FUNCTION F_SCALE_TO_DIOC : A_DIOC_DATA_TYPE
VAR_INPUT
	nValue				: REAL;
	nRAWMin				: REAL;
	nRAWMax				: REAL;
	nSCALEDMin			: REAL;
	nSCALEDMax			: REAL;
	nSCALEDOffset		: REAL;
END_VAR
VAR
END_VAR

F_SCALE_TO_DIOC := TRUNC_INT((nValue - nSCALEDOffset) * (nRAWMax - nRAWMin) / (nSCALEDMax - nSCALEDMin));

END_FUNCTION

// POUs/DIOC/RC/_Internal/FB_DIOC_RC
FUNCTION_BLOCK FB_DIOC_RC
VAR_INPUT
	(* Data handshake interface *)
	test : INT;
	in									: ST_DIOC_RC_IN;
	in_Dioc_Status						: ST_DIOC_OUT;			(* Feedback dioc communication block *)
	in_Dioc_Gen_Status					: ST_DIOC_GEN_OUT;		(* Feedback general registers *)
	(*bDeviceReady						: BOOL;					(* Device charged and ready *)
	bDeviceActive						: BOOL;					(* Device is active *)*)
	Dioc_Register_IN						: ST_DIOC_REGISTER;		(* Message retrieved from buffer *)
END_VAR
VAR_OUTPUT
	(* RC feedback data *)
	out									: ST_DIOC_RC_OUT;
	nError								: E_DIOC_RC_ERROR;
END_VAR
VAR_IN_OUT
	(*Dioc_Register_OUT					: A_DIOC_MESSAGE;*)
	RxBuffer								: ARRAY[0..DIOC_RXTX_BUFFERSIZE] OF A_DIOC_MESSAGE;	(* 1 message queue *)
	TxBuffer								: ARRAY[0..DIOC_MAXPRIORITY, 0..DIOC_RXTX_BUFFERSIZE] OF A_DIOC_MESSAGE;	(* 1 message queue / priority, HIGHEST: 0 = internal priority *)
	(* Fifo Buffer handlers *)
	fbRxBuffer							: FB_DIOC_FIFO;									(* 1 message queue *)
	fbTxBuffer							: ARRAY[0..DIOC_MAXPRIORITY] OF FB_DIOC_FIFO;	(* 1 message queue / priority *)
	(* Restarted ? *)
	bRestarted							: BOOL;
END_VAR
VAR
	(* Previous state in *)
	stDeviceDataInPrevious				: ST_DIOC_RC_IN;

{library private}
	(*
		Timer sync message *)
	tSync								: TON;

	(*
		dioc communication *)
	stDiocRegister						: ST_DIOC_REGISTER;
	stDiocMessage						: A_DIOC_MESSAGE;

	(*
		Sync message response, response is constructed at runtime, can depend on device *)
	dwSyncMessageResponse				: DWORD;

	(*
		device data IN, request to the device *)
	fpDeviceDataInNew					: R_TRIG;

	(*
		Startup list *)
	bStartup							: BOOL 		:= TRUE;

	(* various *)
	i									: INT;
	byToggle							: BYTE;
	nPriority							: INT;		(* This value avoids copy paste errors, filled in by the program, see send action *)
	iRefreshCycles						: INT;

	(* TEMP VARS *)
	nWriteRegister						: A_DIOC_DATA_TYPE;
	(* Buffer read / write *)
	bRxBuffer_Read						: BOOL;
	bRxBuffer_Write						: BOOL;
	bTxBuffer_Read						: BOOL;
	bTxBuffer_Write						: BOOL;

	(* Current values *)
	sR07_UniqueID						: STRING[24];				(* TEMP R7: Unique ID *)
	sR07_UniqueID_hex					: STRING[2];				(* TEMP R7: Unique ID *)
(*
	nR26_Heating_SP						: UINT := 0;				(* R26: Heating 9  SP 0..4095 = 0..10V *)
	nR33_Cooling_SP						: UINT := 0;				(* R33: Cooling 22 SP 0..4095 = 0..10V *)
	nR39_Pulsion_SP						: UINT := 0;				(* R39: RC pulsion 16: 0..10V position command SP 0..4095 = 0..10V *)
	nR45_Extraction_SP					: UINT := 0;				(* R45: RC extraction 29: 0..10V position command SP 0..4095 = 0..10V *)
	nR56_Fan_SP							: UINT := 0;				(* R56: FAN 39-40: 0..10V fanspeed command SP 0..4095 = 0..10V *)*)

	outRef								: ST_DIOC_RC_OUT;


END_VAR

(*startup *)
IF bStartup THEN Startup(); END_IF

(*
	Toggle byte *)
byToggle		:= byToggle + 1;

(* handle restart *)
IF	bRestarted				THEN
	Restart();
END_IF

(*refresh sent data every 1000 cycles*)
IF iRefreshCycles < 1000 THEN
	iRefreshCycles := iRefreshCycles +1;
ELSIF in_Dioc_Gen_Status.nR10_DiocVoltageB > -1 THEN
	iRefreshCycles := 0;
END_IF;

(*Process new data from dioc *)
Receive();

(*External Dioc request processing, with priority handling *)
Send();

(*First loop finished *)
bStartup 					:= FALSE;

ACTION Receive:
(* !!! ONLY ACTIVE WHEN THE DEVICE IS ACTIVE !!! *)

(*New dioc data received and the device is active *)
IF in_Dioc_Status.bRxBufferEmpty	OR NOT in_Dioc_Gen_Status.bDeviceActive THEN
	RETURN;
END_IF

(*
	Process new data *)
CASE Dioc_Register_IN.nRegister			OF

	RC_R20_RC_TEMPERATURE: 				(*20*)
		out.nR20_RCTemperature := F_SCALE_FROM_DIOC(Dioc_Register_IN.nValue, 0, 4095, -20, 120, -20);

	RC_R21_PS_AC_VOLTAGE_LEVEL:			(*21*)
		out.nR21_PsAcVoltageLevel := F_SCALE_FROM_DIOC(Dioc_Register_IN.nValue, 0, 511, 0, 51.1, 0);

	RC_R22_STATUS_BITS_DIPSWITCHES:		(*22*)
		out.bR22_Dipswitch_S01				:= NOT Dioc_Register_IN.nValue.0;
		out.bR22_Dipswitch_S02				:= NOT Dioc_Register_IN.nValue.1;
		out.bR22_Dipswitch_S03				:= NOT Dioc_Register_IN.nValue.2;
		out.bR22_Dipswitch_S04				:= NOT Dioc_Register_IN.nValue.3;
		out.bR22_Dipswitch_S05				:= NOT Dioc_Register_IN.nValue.4;
		out.bR22_Dipswitch_S06				:= NOT Dioc_Register_IN.nValue.5;
		out.bR22_Dipswitch_S07				:= NOT Dioc_Register_IN.nValue.6;
		out.bR22_Dipswitch_S08				:= NOT Dioc_Register_IN.nValue.7;
		out.bR22_Dipswitch_S09				:= NOT Dioc_Register_IN.nValue.8;
		out.bR22_Dipswitch_S10				:= NOT Dioc_Register_IN.nValue.9;
		out.bR22_Dipswitch_S11				:= NOT Dioc_Register_IN.nValue.10;
		out.bR22_Dipswitch_S12				:= NOT Dioc_Register_IN.nValue.11;
		out.sR22_Dipswitch					:= DWORD_TO_BINSTR(Dioc_Register_IN.nValue, 12);

	RC_R25_HEATING_7_8_3P:					(*25*)
		out.bR25_Heating_7_8_3p_plus_pwm	:= NOT Dioc_Register_IN.nValue.0;
		out.bR25_Heating_7_8_3p_min			:= NOT Dioc_Register_IN.nValue.1;

	RC_R26_HEATING_9_SP:					(*26
		out.nR26_HeatingSP 					:= F_SCALE_FROM_DIOC(Dioc_Register_IN.nValue, 0, 4095, 0, 10, 0);*)
		out.nR26_Heating_SP 				:= DWORD_TO_REAL(Dioc_Register_IN.nValue);

	RC_R27_HEATING_12_13_TEMP_HVAC_WATER:	(*27*)
		out.nR27_HeatingTempHvacWater := F_SCALE_FROM_DIOC(Dioc_Register_IN.nValue, 0, 4095, -20, 120, -20);

	RC_R32_COOLING_20_21_3P:				(*32*)
		out.bR32_Cooling_20_21_3p_plus_pwm	:= NOT Dioc_Register_IN.nValue.0;
		out.bR32_Cooling_20_21_3p_min		:= NOT Dioc_Register_IN.nValue.1;

	RC_R33_COOLING_22_SP:					(*33
		out.nR33_CoolingSP 					:= F_SCALE_FROM_DIOC(Dioc_Register_IN.nValue, 0, 4095, 0, 10, 0);*)
		out.nR33_Cooling_SP					:= DWORD_TO_REAL(Dioc_Register_IN.nValue);

	RC_R34_COOLING_25_26_TEMP_ICE_WATER:	(*34*)
		out.nR34_CoolingTempIceWater := F_SCALE_FROM_DIOC(Dioc_Register_IN.nValue, 0, 4095, -20, 120, -20);

	RC_R39_PULSION_16_POSITION_COMMAND:	(*39
		out.nR39_PulsionPositionCOM 		:= F_SCALE_FROM_DIOC(Dioc_Register_IN.nValue, 0, 4095, 0, 10, 0);*)
		out.nR39_Pulsion_SP  				:= DWORD_TO_REAL(Dioc_Register_IN.nValue);

	RC_R40_PULSION_17_POSITION_FEEDBACK:	(*40
		out.nR40_PulsionPositionFB 			:= F_SCALE_FROM_DIOC(Dioc_Register_IN.nValue, 0, 10, 0, 100, 0);*)
		out.nR40_Pulsion_FB := F_SCALE_FROM_DIOC(Dioc_Register_IN.nValue, 0, 4095, 0, 100, 0);

	RC_R42_PULSION_18_AIR_TEMPERATURE:		(*42*)
		out.nR42_PulsionAirTemperature := F_SCALE_FROM_DIOC(Dioc_Register_IN.nValue, 0, 4095, -20, 120, -20);

	RC_R45_EXTRACTION_29_POSITION_COMMAND:	(*45
		out.nR45_ExtractionPositionCOM 		:= F_SCALE_FROM_DIOC(Dioc_Register_IN.nValue, 0, 4095, 0, 10, 0);*)
		out.nR45_Extraction_SP 				:= DWORD_TO_REAL(Dioc_Register_IN.nValue);

	RC_R46_EXTRACTION_30_POSITION_FEEDBACK:(*46
		out.nR46_ExtractionPositionFB 		:= F_SCALE_FROM_DIOC(Dioc_Register_IN.nValue, 0, 10, 0, 100, 0);*)
		out.nR46_Extraction_FB  := F_SCALE_FROM_DIOC(Dioc_Register_IN.nValue, 0, 4095, 0, 100, 0);

	RC_R49_EXTRACTION_31_AIR_TEMPERATURE:	(*49*)
		out.nR49_ExtractionAirTemperature := F_SCALE_FROM_DIOC(Dioc_Register_IN.nValue, 0, 4095, -20, 120, -20);

	RC_R52_FIREDAMPER_33_34_COMMAND:		(*52*)
		out.bR52_FireDamperCOM_NC			:= NOT Dioc_Register_IN.nValue.0;
		out.bR52_FireDamperCOM_NO			:= NOT Dioc_Register_IN.nValue.1;

	RC_R53_FIREDAMPER_36_37_FEEDBACK:		(*53*)
		out.bR53_FireDamperFB_CLS			:= Dioc_Register_IN.nValue.0;
		out.bR53_FireDamperFB_OPN			:= Dioc_Register_IN.nValue.1;

	RC_R56_FAN_39_40_SPEED_COMMAND:		(*56
		out.nR56_FanSpeedCOM 				:= F_SCALE_FROM_DIOC(Dioc_Register_IN.nValue, 0, 4095, 0, 10, 0);*)
		out.nR56_Fan_SP						:= DWORD_TO_REAL(Dioc_Register_IN.nValue);

	RC_R57_FAN_ENABLE:						(*57*)
		out.bR57_Fan_Enable					:= Dioc_Register_IN.nValue.0;

	RC_R58_FAN_FAULT_STATUS:				(*58*)
		out.bR58_FanFaultStatus				:= Dioc_Register_IN.nValue.0;

	RC_R61_DO_45_46_47: 					(*61*)
		out.bR61_do_45				:= Dioc_Register_IN.nValue.2;
		out.bR61_do_46				:= Dioc_Register_IN.nValue.1;
		out.bR61_do_47				:= Dioc_Register_IN.nValue.0;

	ELSE;

END_CASE
END_ACTION

ACTION Restart:
(* Invalidate previous status with something impossible *)
in.bR20_RC_Temperature := NOT stDeviceDataInPrevious.bR20_RC_Temperature;

out := outRef;

(* Acknowledge *)
bRestarted := FALSE;
END_ACTION

ACTION Send:
(* !!! ONLY ACTIVE WHEN THE DEVICE IS ACTIVE !!! *)

(*
	is the device active *)
IF NOT in_Dioc_Gen_Status.bDeviceActive THEN
	RETURN;
END_IF

(*
	Check if a new message is to be sent, confirm by resetting request 
	nR26_HeatingSP						: UINT := 0;				(* R26: Heating 9  SP 0..4095 = 0..10V *)
	nR33_CoolingSP						: UINT := 0;				(* R33: Cooling 22 SP 0..4095 = 0..10V *)
	nR39_PulsionSP						: UINT := 0;				(* R39: RC pulsion 16: 0..10V position command SP 0..4095 = 0..10V *)
	nR45_ExtractionSP					: UINT := 0;				(* R45: RC extraction 29: 0..10V position command SP 0..4095 = 0..10V *)
	nR56_FanspeedSP						: UINT := 0;				(* R56: FAN 39-40: 0..10V fanspeed command SP 0..4095 = 0..10V *)*)
IF in.nR26_Heating_SP <> out.nR26_Heating_SP THEN
	in.bR26_Heating_SP 		:= TRUE;
END_IF
IF in.nR33_Cooling_SP <> out.nR33_Cooling_SP THEN
	in.bR33_Cooling_SP 		:= TRUE;
END_IF
IF in.nR39_Pulsion_SP <> out.nR39_Pulsion_SP THEN
	in.bR39_Pulsion_SP 		:= TRUE;
END_IF
IF in.nR45_Extraction_SP <> out.nR45_Extraction_SP THEN
	in.bR45_Extraction_SP 	:= TRUE;
END_IF
IF in.nR56_Fan_SP <> out.nR56_Fan_SP THEN
	in.bR56_Fan_SP 			:= TRUE;
END_IF

(*
	New dioc data received ? *)
IF MEMCMP(ADR(stDeviceDataInPrevious), ADR(in), SIZEOF(stDeviceDataInPrevious)) = 0 THEN RETURN; END_IF;


(*
	Handle register handling in the order of priority *)
(* PRIORITY 00: internal commands (eg at startup) *)
(* Test message, highest priority, always send a sync message first *)
nPriority := 0;

(* PRIORITY 01 *)
nPriority := 1;

(* PRIORITY 02 *)
nPriority := 2;
(* Register R52_FireDamperCOM_NO / NC *)
IF 	in.bR52_FireDamperCOM_NO  		AND	NOT out.bR52_FireDamperCOM_NO 	OR
	NOT in.bR52_FireDamperCOM_NO 	AND out.bR52_FireDamperCOM_NO 		OR
 	in.bR52_FireDamperCOM_NC  		AND	NOT out.bR52_FireDamperCOM_NC 	OR
	NOT in.bR52_FireDamperCOM_NC 	AND out.bR52_FireDamperCOM_NC 		OR
	iRefreshCycles = 300 THEN
	(* Register value *)
	nWriteRegister					:= 0;
	nWriteRegister.0 				:= in.bR52_FireDamperCOM_NO;
	nWriteRegister.1 				:= in.bR52_FireDamperCOM_NC; (* AND NOT in.bR52_FireDamperCOM_NO;	interlock priority NO *)
	(* Write register *)
	bTxBuffer_Write					:= TRUE;
	fbTxBuffer[nPriority](
		IN							:= F_DIOC_20_MESSAGE_OUT(nRegister := RC_R52_FIREDAMPER_33_34_COMMAND, nValue := nWriteRegister),
		RD							:= bTxBuffer_Read,			(* Not functional *)
		WD							:= bTxBuffer_Write,
		fifo						:= ADR(TxBuffer[nPriority, 0]));	(* Send the register *)
	(* Message buffered? *)
	IF NOT bTxBuffer_Write THEN
		out.bR52_FireDamperCOM_NO							:=
		stDeviceDataInPrevious.bR52_FireDamperCOM_NO 		:= in.bR52_FireDamperCOM_NO;
		out.bR52_FireDamperCOM_NC							:=
		stDeviceDataInPrevious.bR52_FireDamperCOM_NC 		:= in.bR52_FireDamperCOM_NC;
	END_IF
END_IF

(* PRIORITY 03 *)
nPriority := 3;

(* PRIORITY 04 *)
nPriority := 4;

(* PRIORITY 05 *)
nPriority := 5;
(* Register R25_Heating_7_8_3p *)
IF 	in.bR25_Heating_7_8_3p_plus_pwm  	AND	NOT out.bR25_Heating_7_8_3p_plus_pwm 	OR
	NOT in.bR25_Heating_7_8_3p_plus_pwm AND out.bR25_Heating_7_8_3p_plus_pwm 		OR
 	in.bR25_Heating_7_8_3p_min  		AND	NOT out.bR25_Heating_7_8_3p_min		 	OR
	NOT in.bR25_Heating_7_8_3p_min 		AND out.bR25_Heating_7_8_3p_min				OR
	iRefreshCycles = 100 THEN
	(* Register value *)
	nWriteRegister					:= 0;
	nWriteRegister.0 				:= in.bR25_Heating_7_8_3p_plus_pwm;
	nWriteRegister.1 				:= in.bR25_Heating_7_8_3p_min;
	(* Write register *)
	bTxBuffer_Write					:= TRUE;
	fbTxBuffer[nPriority](
		IN							:= F_DIOC_20_MESSAGE_OUT(nRegister := RC_R25_HEATING_7_8_3P, nValue := nWriteRegister),
		RD							:= bTxBuffer_Read,			(* Not functional *)
		WD							:= bTxBuffer_Write,
		fifo						:= ADR(TxBuffer[nPriority, 0]));	(* Send the register *)
	(* Message buffered? *)
	IF NOT bTxBuffer_Write THEN
		out.bR25_Heating_7_8_3p_plus_pwm					:=
		stDeviceDataInPrevious.bR25_Heating_7_8_3p_plus_pwm := in.bR25_Heating_7_8_3p_plus_pwm;
		out.bR25_Heating_7_8_3p_min							:=
		stDeviceDataInPrevious.bR25_Heating_7_8_3p_min 		:= in.bR25_Heating_7_8_3p_min;
		(*in.bR25_Heating_7_8_3p_status := TRUE;*)
	END_IF
END_IF
(* if R25 is not set correctly this code will send it again, but checking R25 doesn't work correctly so this code will spam 25 on the dioc line
IF in.bR25_Heating_7_8_3p_status THEN
	fbTxBuffer[nPriority](
		IN							:= F_DIOC_20_MESSAGE_OUT(nRegister := DIOC_R01_REGISTER_REQUEST, nValue := RC_R25_HEATING_7_8_3P),
		RD							:= bTxBuffer_Read,			(* Not functional *)
		WD							:= in.bR25_Heating_7_8_3p_status,
		fifo						:= ADR(TxBuffer[nPriority, 0]));
	in.bR25_Heating_7_8_3p_status := FALSE;
END_IF*)

(* Register R32_Cooling_20_21_3p *)
IF 	in.bR32_Cooling_20_21_3p_plus_pwm  	AND	NOT out.bR32_Cooling_20_21_3p_plus_pwm 	OR
	NOT in.bR32_Cooling_20_21_3p_plus_pwm AND out.bR32_Cooling_20_21_3p_plus_pwm 	OR
 	in.bR32_Cooling_20_21_3p_min  		AND	NOT out.bR32_Cooling_20_21_3p_min		OR
	NOT in.bR32_Cooling_20_21_3p_min 	AND out.bR32_Cooling_20_21_3p_min			OR
	iRefreshCycles = 200 THEN
	(* Register value *)
	nWriteRegister					:= 0;
	nWriteRegister.0 				:= in.bR32_Cooling_20_21_3p_plus_pwm;
	nWriteRegister.1 				:= in.bR32_Cooling_20_21_3p_min;
	(* Write register *)
	bTxBuffer_Write					:= TRUE;
	fbTxBuffer[nPriority](
		IN							:= F_DIOC_20_MESSAGE_OUT(nRegister := RC_R32_COOLING_20_21_3P, nValue := nWriteRegister),
		RD							:= bTxBuffer_Read,			(* Not functional *)
		WD							:= bTxBuffer_Write,
		fifo						:= ADR(TxBuffer[nPriority, 0]));	(* Send the register *)
	(* Message buffered? *)
	IF NOT bTxBuffer_Write THEN
		out.bR32_Cooling_20_21_3p_plus_pwm						:=
		stDeviceDataInPrevious.bR32_Cooling_20_21_3p_plus_pwm 	:= in.bR32_Cooling_20_21_3p_plus_pwm;
		out.bR32_Cooling_20_21_3p_min							:=
		stDeviceDataInPrevious.bR32_Cooling_20_21_3p_min 		:= in.bR32_Cooling_20_21_3p_min;
	END_IF
END_IF
(* Register R57_FAN_Enable_command *)
IF 	in.bR57_Fan_Enable 	AND	NOT out.bR57_Fan_Enable 	OR
	NOT in.bR57_Fan_Enable AND out.bR57_Fan_Enable OR
	iRefreshCycles = 400 	THEN
	(* Register value *)
	nWriteRegister					:= 0;
	nWriteRegister.0 				:= in.bR57_Fan_Enable;
	(* Write register *)
	bTxBuffer_Write					:= TRUE;
	fbTxBuffer[nPriority](
		IN							:= F_DIOC_20_MESSAGE_OUT(nRegister := RC_R57_FAN_ENABLE, nValue := nWriteRegister),
		RD							:= bTxBuffer_Read,			(* Not functional *)
		WD							:= bTxBuffer_Write,
		fifo						:= ADR(TxBuffer[nPriority, 0]));	(* Send the register *)
	(* Message buffered? *)
	IF NOT bTxBuffer_Write THEN
		out.bR57_Fan_Enable						:=
		stDeviceDataInPrevious.bR57_Fan_Enable 	:= in.bR57_Fan_Enable;
	END_IF
END_IF

IF (in.bR61_do_45 AND NOT  out.bR61_do_45)
	OR (NOT in.bR61_do_45 AND out.bR61_do_45)
	OR (in.bR61_do_46 AND NOT  out.bR61_do_46)
	OR (NOT in.bR61_do_46 AND out.bR61_do_46)
	OR (in.bR61_do_47 AND NOT  out.bR61_do_47)
	OR (NOT in.bR61_do_47 AND out.bR61_do_47)OR
	iRefreshCycles = 600  THEN
(* Register value *)
	nWriteRegister					:= 0;
	nWriteRegister.0 				:= in.bR61_do_47;
	nWriteRegister.1 				:= in.bR61_do_46;
	nWriteRegister.2 				:= in.bR61_do_45;
	(* Write register *)
	bTxBuffer_Write					:= TRUE;
	fbTxBuffer[nPriority](
		IN							:= F_DIOC_20_MESSAGE_OUT(nRegister := RC_R61_DO_45_46_47, nValue := nWriteRegister),
		RD							:= bTxBuffer_Read,			(* Not functional *)
		WD							:= bTxBuffer_Write,
		fifo						:= ADR(TxBuffer[nPriority, 0]));
	IF NOT bTxBuffer_Write THEN
		out.bR61_do_45 		:= stDeviceDataInPrevious.bR61_do_45	 	:= in.bR61_do_45;
		out.bR61_do_46 		:= stDeviceDataInPrevious.bR61_do_46 		:= in.bR61_do_46;
		out.bR61_do_47 		:= stDeviceDataInPrevious.bR61_do_47		:= in.bR61_do_47;
	END_IF
END_IF

(* PRIORITY 06 *)
nPriority := 6;
IF in.bR26_Heating_SP THEN
	out.nR26_Heating_SP				:= -1;
	fbTxBuffer[nPriority](
		IN							:= F_DIOC_20_MESSAGE_OUT(nRegister := RC_R26_HEATING_9_SP, nValue := in.nR26_Heating_SP),
		RD							:= bTxBuffer_Read,			(* Not functional *)
		WD							:= in.bR26_Heating_SP,
		fifo						:= ADR(TxBuffer[nPriority, 0]));
	IF NOT in.bR26_Heating_SP		THEN 	out.nR26_Heating_SP := in.nR26_Heating_SP; END_IF
END_IF
IF in.bR33_Cooling_SP THEN
	out.nR33_Cooling_SP				:= -1;
	fbTxBuffer[nPriority](
		IN							:= F_DIOC_20_MESSAGE_OUT(nRegister := RC_R33_COOLING_22_SP, nValue := in.nR33_Cooling_SP),
		RD							:= bTxBuffer_Read,			(* Not functional *)
		WD							:= in.bR33_Cooling_SP,
		fifo						:= ADR(TxBuffer[nPriority, 0]));
	IF NOT in.bR33_Cooling_SP		THEN 	out.nR33_Cooling_SP := in.nR33_Cooling_SP; END_IF
END_IF
IF in.bR39_Pulsion_SP THEN
	out.nR39_Pulsion_SP				:= -1;
	fbTxBuffer[nPriority](
		IN							:= F_DIOC_20_MESSAGE_OUT(nRegister := RC_R39_PULSION_16_POSITION_COMMAND, nValue := in.nR39_Pulsion_SP),
		RD							:= bTxBuffer_Read,			(* Not functional *)
		WD							:= in.bR39_Pulsion_SP,
		fifo						:= ADR(TxBuffer[nPriority, 0]));
	IF NOT in.bR39_Pulsion_SP		THEN 	out.nR39_Pulsion_SP := in.nR39_Pulsion_SP; END_IF
END_IF
IF in.bR45_Extraction_SP THEN
	out.nR45_Extraction_SP			:= -1;
	fbTxBuffer[nPriority](
		IN							:= F_DIOC_20_MESSAGE_OUT(nRegister := RC_R45_EXTRACTION_29_POSITION_COMMAND, nValue := in.nR45_Extraction_SP),
		RD							:= bTxBuffer_Read,			(* Not functional *)
		WD							:= in.bR45_Extraction_SP,
		fifo						:= ADR(TxBuffer[nPriority, 0]));
	IF NOT in.bR45_Extraction_SP	THEN 	out.nR45_Extraction_SP := in.nR45_Extraction_SP; END_IF
END_IF
IF in.bR56_Fan_SP THEN
	out.nR56_Fan_SP					:= -1;
	fbTxBuffer[nPriority](
		IN							:= F_DIOC_20_MESSAGE_OUT(nRegister := RC_R56_FAN_39_40_SPEED_COMMAND, nValue := in.nR56_Fan_SP),
		RD							:= bTxBuffer_Read,			(* Not functional *)
		WD							:= in.bR56_Fan_SP,
		fifo						:= ADR(TxBuffer[nPriority, 0]));
	IF NOT in.bR56_Fan_SP			THEN 	out.nR56_Fan_SP := in.nR56_Fan_SP; END_IF
END_IF


(* PRIORITY 07 *)
nPriority := 7;


